C09138=1192.956,372.415,-78.592,-176.020,8.369,148.494
C09139=1192.960,372.168,-78.558,-176.022,8.366,148.494
C09140=1192.964,371.920,-78.523,-176.023,8.362,148.493
C09141=1192.968,371.672,-78.490,-176.024,8.359,148.493
C09142=1192.973,371.425,-78.456,-176.026,8.355,148.492
C09143=1192.976,371.177,-78.422,-176.027,8.353,148.492
C09144=1192.981,370.930,-78.387,-176.029,8.349,148.491
C09145=1192.985,370.683,-78.353,-176.030,8.346,148.491
C09146=1192.989,370.434,-78.318,-176.032,8.342,148.490
C09147=1192.993,370.187,-78.285,-176.033,8.339,148.490
C09148=1192.997,369.939,-78.251,-176.035,8.336,148.490
C09149=1193.000,369.692,-78.217,-176.036,8.333,148.489
C09150=1193.005,369.444,-78.182,-176.038,8.329,148.489
C09151=1193.009,369.196,-78.149,-176.039,8.327,148.488
C09152=1193.013,368.948,-78.114,-176.041,8.323,148.488
C09153=1193.017,368.701,-78.080,-176.042,8.320,148.488
C09154=1193.021,368.454,-78.046,-176.044,8.317,148.487
C09155=1193.025,368.205,-78.012,-176.045,8.314,148.487
C09156=1193.029,367.958,-77.978,-176.047,8.310,148.486
C09157=1193.033,367.711,-77.944,-176.048,8.307,148.486
C09158=1193.037,367.462,-77.910,-176.050,8.304,148.485
C09159=1193.042,367.215,-77.876,-176.051,8.300,148.485
C09160=1193.045,366.968,-77.842,-176.053,8.297,148.485
C09161=1193.050,366.686,-77.804,-176.054,8.294,148.484
C09162=1193.055,366.405,-77.765,-176.056,8.290,148.484
C09163=1193.059,366.125,-77.727,-176.059,8.285,148.483
C09164=1193.063,365.843,-77.688,-176.060,8.282,148.483
C09165=1193.068,365.596,-77.655,-176.062,8.279,148.482
C09166=1193.072,365.348,-77.620,-176.063,8.275,148.482
C09167=1193.075,365.100,-77.586,-176.065,8.272,148.482
C09168=1193.080,364.853,-77.553,-176.066,8.269,148.481
C09169=1193.084,364.605,-77.519,-176.069,8.266,148.481
C09170=1193.088,364.357,-77.485,-176.070,8.262,148.481
C09171=1193.092,364.110,-77.451,-176.072,8.259,148.480
C09172=1193.096,363.862,-77.417,-176.074,8.256,148.480
C09173=1193.100,363.615,-77.384,-176.075,8.252,148.479
C09174=1193.104,363.367,-77.350,-176.077,8.249,148.479
C09175=1193.108,363.119,-77.316,-176.079,8.246,148.479
C09176=1193.112,362.871,-77.282,-176.081,8.242,148.478
C09177=1193.116,362.624,-77.249,-176.082,8.240,148.478
C09178=1193.120,362.376,-77.215,-176.084,8.236,148.478
C09179=1193.124,362.129,-77.182,-176.086,8.232,148.477
C09180=1193.129,361.880,-77.147,-176.088,8.229,148.477
C09181=1193.133,361.633,-77.114,-176.089,8.226,148.477
C09182=1193.136,361.385,-77.080,-176.091,8.223,148.476
C09183=1193.141,361.138,-77.047,-176.093,8.219,148.476
C09184=1193.145,360.890,-77.013,-176.095,8.217,148.476
C09185=1193.149,360.642,-76.979,-176.096,8.213,148.475
C09186=1193.153,360.394,-76.946,-176.099,8.210,148.475
C09187=1193.157,360.147,-76.912,-176.100,8.206,148.474
C09188=1193.161,359.899,-76.879,-176.103,8.203,148.474
C09189=1193.166,359.651,-76.845,-176.104,8.200,148.474
C09190=1193.169,359.403,-76.811,-176.106,8.196,148.473
C09191=1193.173,359.156,-76.778,-176.108,8.193,148.473
C09192=1193.177,358.908,-76.745,-176.110,8.189,148.473
C09193=1193.181,358.660,-76.712,-176.111,8.187,148.473
C09194=1193.185,358.413,-76.678,-176.113,8.183,148.472
C09195=1193.189,358.165,-76.645,-176.115,8.180,148.472
C09196=1193.194,357.917,-76.611,-176.118,8.176,148.472
C09197=1193.198,357.669,-76.577,-176.119,8.173,148.471
C09198=1193.202,357.422,-76.543,-176.121,8.170,148.471
C09199=1193.206,357.174,-76.510,-176.123,8.167,148.471
C09200=1193.210,356.926,-76.477,-176.125,8.163,148.470
C09201=1193.214,356.679,-76.444,-176.127,8.160,148.470
C09202=1193.218,356.431,-76.411,-176.129,8.156,148.470
C09203=1193.222,356.183,-76.378,-176.131,8.154,148.470
C09204=1193.226,355.936,-76.344,-176.133,8.150,148.469
C09205=1193.230,355.688,-76.310,-176.135,8.147,148.469
C09206=1193.234,355.440,-76.277,-176.137,8.143,148.468
C09207=1193.239,355.192,-76.243,-176.139,8.140,148.468
C09208=1193.243,354.944,-76.210,-176.141,8.137,148.468
C09209=1193.247,354.696,-76.177,-176.142,8.134,148.468
C09210=1193.251,354.449,-76.144,-176.145,8.131,148.467
C09211=1193.255,354.201,-76.111,-176.147,8.127,148.467
C09212=1193.259,353.953,-76.078,-176.149,8.124,148.467
C09213=1193.263,353.705,-76.044,-176.151,8.120,148.466
C09214=1193.268,353.458,-76.011,-176.153,8.118,148.466
C09215=1193.272,353.210,-75.978,-176.155,8.114,148.466
C09216=1193.276,352.962,-75.945,-176.157,8.111,148.466
C09217=1193.280,352.715,-75.912,-176.159,8.107,148.465
C09218=1193.284,352.467,-75.879,-176.161,8.104,148.465
C09219=1193.288,352.219,-75.846,-176.163,8.102,148.465
C09220=1193.292,351.972,-75.813,-176.165,8.098,148.465
C09221=1193.296,351.724,-75.780,-176.167,8.095,148.464
C09222=1193.300,351.476,-75.747,-176.169,8.091,148.464
C09223=1193.304,351.228,-75.713,-176.171,8.088,148.464
C09224=1193.308,350.981,-75.680,-176.173,8.086,148.464
C09225=1193.312,350.733,-75.647,-176.175,8.082,148.464
C09226=1193.317,350.485,-75.614,-176.177,8.079,148.463
C09227=1193.321,350.237,-75.582,-176.179,8.075,148.463
C09228=1193.325,349.989,-75.548,-176.181,8.072,148.463
C09229=1193.329,349.741,-75.515,-176.184,8.069,148.462
C09230=1193.333,349.494,-75.482,-176.185,8.066,148.462
C09231=1193.337,349.246,-75.450,-176.188,8.063,148.462
C09232=1193.341,348.999,-75.416,-176.190,8.059,148.462
C09233=1193.345,348.750,-75.384,-176.192,8.056,148.461
C09234=1193.350,348.503,-75.351,-176.194,8.052,148.461
C09235=1193.354,348.255,-75.318,-176.195,8.050,148.461
C09236=1193.358,348.007,-75.284,-176.198,8.047,148.461
C09237=1193.362,347.759,-75.252,-176.200,8.043,148.461
C09238=1193.366,347.511,-75.219,-176.202,8.040,148.460
C09239=1193.370,347.264,-75.186,-176.204,8.037,148.460
C09240=1193.374,347.016,-75.153,-176.207,8.033,148.460
C09241=1193.378,346.768,-75.121,-176.208,8.031,148.460
C09242=1193.383,346.520,-75.088,-176.211,8.027,148.459
C09243=1193.386,346.272,-75.055,-176.213,8.024,148.459
C09244=1193.390,346.024,-75.023,-176.215,8.021,148.459
C09245=1193.395,345.777,-74.990,-176.217,8.017,148.459
C09246=1193.400,345.529,-74.957,-176.219,8.015,148.459
C09247=1193.403,345.281,-74.925,-176.221,8.012,148.458
C09248=1193.407,345.033,-74.892,-176.223,8.008,148.458
C09249=1193.412,344.785,-74.859,-176.226,8.005,148.458
C09250=1193.416,344.537,-74.826,-176.228,8.002,148.458
C09251=1193.419,344.289,-74.794,-176.230,7.998,148.458
C09252=1193.423,344.042,-74.761,-176.232,7.996,148.457
C09253=1193.428,343.793,-74.729,-176.234,7.993,148.457
C09254=1193.432,343.547,-74.696,-176.236,7.989,148.457
C09255=1193.436,343.298,-74.664,-176.239,7.986,148.457
C09256=1193.441,343.050,-74.631,-176.241,7.983,148.456
C09257=1193.445,342.802,-74.598,-176.242,7.980,148.456
C09258=1193.448,342.555,-74.566,-176.245,7.977,148.456
C09259=1193.453,342.306,-74.533,-176.247,7.973,148.456
C09260=1193.458,342.059,-74.501,-176.250,7.970,148.456
C09261=1193.461,341.811,-74.469,-176.252,7.967,148.456
C09262=1193.465,341.564,-74.436,-176.254,7.965,148.455
C09263=1193.469,341.316,-74.404,-176.256,7.961,148.455
C09264=1193.473,341.068,-74.371,-176.258,7.958,148.455
C09265=1193.478,340.789,-74.335,-176.260,7.955,148.455
C09266=1193.483,340.511,-74.299,-176.263,7.950,148.455
C09267=1193.488,340.232,-74.262,-176.266,7.947,148.455
C09268=1193.492,339.954,-74.225,-176.268,7.944,148.454
C09269=1193.496,339.705,-74.193,-176.270,7.941,148.454
C09270=1193.500,339.457,-74.161,-176.272,7.937,148.454
C09271=1193.504,339.210,-74.128,-176.275,7.934,148.454
C09272=1193.509,338.962,-74.096,-176.277,7.931,148.454
C09273=1193.513,338.714,-74.064,-176.279,7.929,148.453
C09274=1193.517,338.466,-74.031,-176.281,7.925,148.453
C09275=1193.521,338.218,-73.999,-176.284,7.922,148.453
C09276=1193.526,337.970,-73.967,-176.286,7.919,148.453
C09277=1193.530,337.722,-73.935,-176.288,7.916,148.453
C09278=1193.534,337.475,-73.902,-176.290,7.913,148.453
C09279=1193.537,337.227,-73.870,-176.292,7.910,148.452
C09280=1193.543,336.979,-73.838,-176.295,7.906,148.452
C09281=1193.546,336.731,-73.806,-176.297,7.903,148.452
C09282=1193.551,336.483,-73.774,-176.300,7.900,148.452
C09283=1193.554,336.235,-73.742,-176.301,7.898,148.452
C09284=1193.558,335.988,-73.710,-176.303,7.894,148.452
C09285=1193.563,335.739,-73.677,-176.306,7.891,148.452
C09286=1193.567,335.491,-73.645,-176.308,7.888,148.451
C09287=1193.571,335.243,-73.613,-176.311,7.885,148.451
C09288=1193.575,334.996,-73.581,-176.313,7.882,148.451
C09289=1193.580,334.747,-73.549,-176.315,7.879,148.451
C09290=1193.583,334.499,-73.517,-176.317,7.876,148.451
C09291=1193.588,334.252,-73.486,-176.320,7.872,148.451
C09292=1193.592,334.004,-73.453,-176.322,7.869,148.451
C09293=1193.596,333.756,-73.421,-176.324,7.866,148.450
C09294=1193.600,333.508,-73.390,-176.326,7.864,148.450
C09295=1193.605,333.260,-73.358,-176.329,7.860,148.450
C09296=1193.608,333.012,-73.326,-176.331,7.857,148.450
C09297=1193.613,332.764,-73.294,-176.334,7.854,148.450
C09298=1193.617,332.516,-73.262,-176.336,7.851,148.450
C09299=1193.621,332.268,-73.230,-176.338,7.848,148.450
C09300=1193.626,332.021,-73.198,-176.340,7.845,148.450
C09301=1193.630,331.773,-73.166,-176.343,7.842,148.449
C09302=1193.633,331.524,-73.134,-176.345,7.839,148.449
C09303=1193.638,331.277,-73.103,-176.348,7.836,148.449
C09304=1193.642,331.029,-73.070,-176.349,7.833,148.449
C09305=1193.646,330.781,-73.038,-176.352,7.830,148.449
C09306=1193.650,330.533,-73.007,-176.354,7.827,148.449
C09307=1193.654,330.285,-72.974,-176.356,7.823,148.449
C09308=1193.659,330.037,-72.944,-176.359,7.820,148.449
C09309=1193.663,329.789,-72.912,-176.361,7.817,148.448
C09310=1193.666,329.541,-72.880,-176.363,7.815,148.448
C09311=1193.672,329.293,-72.848,-176.366,7.812,148.448
C09312=1193.675,329.045,-72.816,-176.368,7.809,148.448
C09313=1193.680,328.797,-72.785,-176.371,7.805,148.448
C09314=1193.684,328.549,-72.753,-176.373,7.802,148.448
C09315=1193.687,328.301,-72.722,-176.375,7.800,148.448
C09316=1193.692,328.054,-72.690,-176.377,7.796,148.448
C09317=1193.696,327.805,-72.658,-176.380,7.793,148.448
C09318=1193.701,327.558,-72.627,-176.382,7.790,148.447
C09319=1193.704,327.310,-72.595,-176.385,7.787,148.447
C09320=1193.709,327.062,-72.564,-176.387,7.785,148.447
C09321=1193.713,326.814,-72.532,-176.389,7.782,148.447
C09322=1193.718,326.566,-72.500,-176.391,7.778,148.447
C09323=1193.721,326.318,-72.469,-176.394,7.775,148.447
C09324=1193.725,326.069,-72.437,-176.396,7.772,148.447
C09325=1193.730,325.822,-72.406,-176.399,7.770,148.447
C09326=1193.734,325.573,-72.375,-176.401,7.766,148.447
C09327=1193.738,325.326,-72.343,-176.403,7.763,148.447
C09328=1193.742,325.078,-72.311,-176.406,7.760,148.446
C09329=1193.746,324.830,-72.281,-176.408,7.757,148.446
C09330=1193.750,324.582,-72.249,-176.410,7.754,148.446
C09331=1193.755,324.334,-72.218,-176.413,7.751,148.446
C09332=1193.759,324.086,-72.186,-176.415,7.748,148.446
C09333=1193.764,323.838,-72.155,-176.418,7.745,148.446
C09334=1193.767,323.590,-72.123,-176.420,7.743,148.446
C09335=1193.772,323.342,-72.092,-176.422,7.740,148.446
C09336=1193.776,323.094,-72.060,-176.425,7.737,148.446
C09337=1193.780,322.846,-72.029,-176.427,7.733,148.446
C09338=1193.784,322.598,-71.998,-176.430,7.730,148.446
C09339=1193.789,322.350,-71.967,-176.432,7.728,148.446
C09340=1193.792,322.102,-71.935,-176.434,7.725,148.446
C09341=1193.797,321.854,-71.904,-176.437,7.722,148.446
C09342=1193.801,321.606,-71.873,-176.439,7.718,148.445
C09343=1193.805,321.358,-71.842,-176.442,7.715,148.445
C09344=1193.810,321.110,-71.810,-176.444,7.713,148.445
C09345=1193.814,320.862,-71.779,-176.446,7.710,148.445
C09346=1193.818,320.614,-71.749,-176.449,7.707,148.445
C09347=1193.821,320.366,-71.717,-176.451,7.704,148.445
C09348=1193.826,320.118,-71.686,-176.453,7.701,148.445
C09349=1193.830,319.869,-71.655,-176.456,7.698,148.445
C09350=1193.834,319.622,-71.624,-176.458,7.695,148.445
C09351=1193.839,319.374,-71.593,-176.461,7.692,148.445
C09352=1193.843,319.125,-71.562,-176.464,7.689,148.445
C09353=1193.847,318.878,-71.531,-176.465,7.686,148.445
C09354=1193.851,318.629,-71.499,-176.468,7.683,148.445
C09355=1193.856,318.381,-71.469,-176.470,7.680,148.444
C09356=1193.860,318.133,-71.438,-176.473,7.677,148.444
C09357=1193.864,317.885,-71.407,-176.476,7.674,148.444
C09358=1193.868,317.638,-71.376,-176.477,7.672,148.444
C09359=1193.873,317.390,-71.345,-176.480,7.669,148.444
C09360=1193.877,317.141,-71.314,-176.483,7.666,148.444
C09361=1193.881,316.893,-71.283,-176.485,7.663,148.444
C09362=1193.885,316.645,-71.252,-176.487,7.660,148.444
C09363=1193.889,316.398,-71.221,-176.490,7.657,148.444
C09364=1193.893,316.150,-71.190,-176.492,7.654,148.444
C09365=1193.897,315.901,-71.159,-176.495,7.651,148.444
C09366=1193.902,315.653,-71.129,-176.497,7.649,148.444
C09367=1193.907,315.405,-71.098,-176.499,7.645,148.444
C09368=1193.910,315.157,-71.067,-176.502,7.642,148.444
C09369=1193.915,314.881,-71.032,-176.504,7.639,148.444
C09370=1193.920,314.603,-70.998,-176.507,7.636,148.444
C09371=1193.925,314.328,-70.964,-176.510,7.632,148.444
C09372=1193.929,314.052,-70.930,-176.513,7.629,148.444
C09373=1193.933,313.803,-70.899,-176.515,7.626,148.444
C09374=1193.937,313.556,-70.869,-176.517,7.624,148.444
C09375=1193.942,313.308,-70.838,-176.520,7.621,148.444
C09376=1193.946,313.059,-70.807,-176.523,7.618,148.444
C09377=1193.951,312.811,-70.776,-176.525,7.614,148.444
C09378=1193.954,312.563,-70.746,-176.527,7.612,148.444
C09379=1193.959,312.315,-70.715,-176.530,7.609,148.444
C09380=1193.963,312.067,-70.684,-176.533,7.606,148.444
C09381=1193.967,311.818,-70.654,-176.535,7.603,148.443
C09382=1193.972,311.570,-70.624,-176.537,7.601,148.443
C09383=1193.976,311.323,-70.593,-176.540,7.598,148.443
C09384=1193.980,311.074,-70.562,-176.542,7.595,148.443
C09385=1193.984,310.826,-70.532,-176.545,7.591,148.443
C09386=1193.988,310.579,-70.501,-176.547,7.589,148.443
C09387=1193.993,310.331,-70.471,-176.549,7.586,148.443
C09388=1193.997,310.082,-70.439,-176.552,7.583,148.443
C09389=1194.001,309.834,-70.410,-176.555,7.580,148.443
C09390=1194.006,309.586,-70.379,-176.557,7.578,148.443
C09391=1194.010,309.338,-70.349,-176.559,7.575,148.443
C09392=1194.014,309.090,-70.318,-176.562,7.572,148.443
C09393=1194.018,308.841,-70.288,-176.565,7.569,148.443
C09394=1194.022,308.593,-70.258,-176.567,7.566,148.443
C09395=1194.027,308.345,-70.227,-176.569,7.563,148.443
C09396=1194.031,308.098,-70.197,-176.572,7.560,148.443
C09397=1194.036,307.849,-70.167,-176.574,7.557,148.443
C09398=1194.039,307.601,-70.136,-176.577,7.555,148.443
C09399=1194.044,307.353,-70.105,-176.579,7.552,148.443
C09400=1194.048,307.104,-70.076,-176.582,7.549,148.443
C09401=1194.052,306.856,-70.045,-176.584,7.545,148.443
C09402=1194.056,306.609,-70.015,-176.586,7.543,148.443
C09403=1194.061,306.360,-69.985,-176.589,7.540,148.443
C09404=1194.065,306.113,-69.955,-176.592,7.537,148.443
C09405=1194.069,305.864,-69.924,-176.594,7.534,148.443
C09406=1194.073,305.616,-69.894,-176.597,7.532,148.443
C09407=1194.078,305.368,-69.864,-176.599,7.529,148.443
C09408=1194.082,305.119,-69.834,-176.602,7.526,148.443
C09409=1194.087,304.871,-69.803,-176.604,7.524,148.443
C09410=1194.091,304.623,-69.774,-176.606,7.521,148.443
C09411=1194.095,304.375,-69.743,-176.609,7.518,148.443
C09412=1194.099,304.128,-69.713,-176.612,7.515,148.443
C09413=1194.104,303.879,-69.683,-176.614,7.512,148.443
C09414=1194.108,303.631,-69.652,-176.617,7.509,148.443
C09415=1194.112,303.382,-69.623,-176.619,7.506,148.443
C09416=1194.116,303.134,-69.592,-176.622,7.503,148.443
C09417=1194.121,302.886,-69.563,-176.624,7.501,148.443
C09418=1194.125,302.638,-69.533,-176.626,7.498,148.443
C09419=1194.129,302.390,-69.502,-176.629,7.495,148.443
C09420=1194.134,302.142,-69.473,-176.631,7.493,148.443
C09421=1194.137,301.894,-69.443,-176.634,7.490,148.443
C09422=1194.142,301.645,-69.413,-176.637,7.487,148.443
C09423=1194.146,301.397,-69.383,-176.639,7.484,148.443
C09424=1194.150,301.150,-69.353,-176.642,7.481,148.443
C09425=1194.155,300.901,-69.323,-176.644,7.478,148.443
C09426=1194.159,300.653,-69.293,-176.647,7.475,148.443
C09427=1194.163,300.405,-69.263,-176.649,7.473,148.443
C09428=1194.168,300.156,-69.233,-176.651,7.470,148.443
C09429=1194.172,299.908,-69.204,-176.654,7.467,148.443
C09430=1194.176,299.661,-69.174,-176.656,7.465,148.443
C09431=1194.180,299.412,-69.144,-176.659,7.462,148.443
C09432=1194.185,299.164,-69.114,-176.662,7.459,148.443
C09433=1194.189,298.916,-69.084,-176.664,7.456,148.443
C09434=1194.193,298.668,-69.055,-176.666,7.453,148.443
C09435=1194.198,298.420,-69.025,-176.669,7.450,148.443
C09436=1194.203,298.171,-68.995,-176.672,7.447,148.443
C09437=1194.206,297.923,-68.965,-176.674,7.445,148.444
C09438=1194.211,297.675,-68.936,-176.677,7.442,148.444
C09439=1194.215,297.427,-68.906,-176.679,7.439,148.444
C09440=1194.219,297.179,-68.877,-176.682,7.437,148.444
C09441=1194.224,296.930,-68.847,-176.684,7.434,148.444
C09442=1194.228,296.682,-68.817,-176.687,7.431,148.444
C09443=1194.232,296.434,-68.787,-176.690,7.428,148.444
C09444=1194.236,296.186,-68.758,-176.692,7.426,148.444
C09445=1194.240,295.938,-68.728,-176.694,7.423,148.444
C09446=1194.245,295.689,-68.699,-176.697,7.420,148.444
C09447=1194.249,295.441,-68.669,-176.699,7.418,148.444
C09448=1194.254,295.192,-68.639,-176.702,7.415,148.444
C09449=1194.258,294.944,-68.610,-176.705,7.412,148.444
C09450=1194.262,294.696,-68.580,-176.707,7.409,148.444
C09451=1194.266,294.448,-68.551,-176.710,7.406,148.444
C09452=1194.270,294.199,-68.521,-176.712,7.403,148.444
C09453=1194.275,293.952,-68.492,-176.714,7.401,148.444
C09454=1194.279,293.703,-68.463,-176.717,7.398,148.444
C09455=1194.283,293.455,-68.433,-176.720,7.395,148.444
C09456=1194.288,293.207,-68.404,-176.722,7.393,148.444
C09457=1194.292,292.959,-68.374,-176.725,7.390,148.444
C09458=1194.296,292.710,-68.345,-176.727,7.387,148.444
C09459=1194.300,292.462,-68.316,-176.730,7.385,148.444
C09460=1194.304,292.214,-68.286,-176.732,7.382,148.444
C09461=1194.309,291.966,-68.257,-176.735,7.379,148.444
C09462=1194.313,291.718,-68.228,-176.737,7.377,148.444
C09463=1194.318,291.470,-68.198,-176.740,7.374,148.444
C09464=1194.322,291.221,-68.169,-176.743,7.371,148.444
C09465=1194.326,290.973,-68.140,-176.745,7.369,148.445
C09466=1194.330,290.724,-68.110,-176.747,7.365,148.445
C09467=1194.335,290.476,-68.081,-176.750,7.362,148.445
C09468=1194.339,290.229,-68.052,-176.752,7.360,148.445
C09469=1194.344,289.980,-68.022,-176.755,7.357,148.445
C09470=1194.348,289.731,-67.994,-176.758,7.354,148.445
C09471=1194.352,289.483,-67.964,-176.760,7.352,148.445
C09472=1194.356,289.235,-67.935,-176.763,7.349,148.445
C09473=1194.361,288.960,-67.903,-176.765,7.346,148.445
C09474=1194.366,288.686,-67.870,-176.768,7.343,148.445
C09475=1194.371,288.411,-67.838,-176.771,7.340,148.445
C09476=1194.375,288.137,-67.807,-176.774,7.337,148.445
C09477=1194.380,287.889,-67.777,-176.777,7.334,148.445
C09478=1194.384,287.640,-67.748,-176.779,7.332,148.445
C09479=1194.389,287.392,-67.719,-176.781,7.329,148.445
C09480=1194.393,287.144,-67.690,-176.784,7.326,148.445
C09481=1194.397,286.896,-67.660,-176.786,7.324,148.445
C09482=1194.401,286.647,-67.632,-176.789,7.321,148.445
C09483=1194.406,286.400,-67.603,-176.792,7.318,148.446
C09484=1194.410,286.151,-67.574,-176.794,7.316,148.446
C09485=1194.414,285.902,-67.545,-176.797,7.313,148.446
C09486=1194.419,285.654,-67.515,-176.799,7.311,148.446
C09487=1194.424,285.406,-67.487,-176.802,7.308,148.446
C09488=1194.427,285.158,-67.458,-176.805,7.305,148.446
C09489=1194.432,284.909,-67.430,-176.807,7.303,148.446
C09490=1194.436,284.662,-67.400,-176.809,7.300,148.446
C09491=1194.441,284.413,-67.371,-176.812,7.297,148.446
C09492=1194.444,284.165,-67.343,-176.814,7.295,148.446
C09493=1194.449,283.916,-67.313,-176.817,7.292,148.446
C09494=1194.454,283.668,-67.285,-176.820,7.290,148.446
C09495=1194.458,283.419,-67.256,-176.822,7.287,148.446
C09496=1194.462,283.171,-67.227,-176.825,7.284,148.446
C09497=1194.467,282.923,-67.199,-176.827,7.282,148.447
C09498=1194.471,282.675,-67.170,-176.830,7.279,148.447
C09499=1194.475,282.426,-67.141,-176.832,7.276,148.447
C09500=1194.479,282.179,-67.112,-176.835,7.273,148.447
C09501=1194.484,281.930,-67.084,-176.838,7.271,148.447
C09502=1194.488,281.681,-67.055,-176.840,7.268,148.447
C09503=1194.492,281.434,-67.026,-176.843,7.265,148.447
C09504=1194.497,281.185,-66.998,-176.845,7.262,148.447
C09505=1194.501,280.937,-66.968,-176.848,7.260,148.447
C09506=1194.505,280.689,-66.940,-176.850,7.257,148.447
C09507=1194.510,280.440,-66.912,-176.852,7.255,148.447
C09508=1194.514,280.192,-66.882,-176.856,7.252,148.447
C09509=1194.518,279.944,-66.854,-176.858,7.249,148.448
C09510=1194.523,279.695,-66.826,-176.860,7.247,148.448
C09511=1194.527,279.447,-66.798,-176.863,7.244,148.448
C09512=1194.531,279.199,-66.768,-176.865,7.242,148.448
C09513=1194.536,278.950,-66.740,-176.868,7.239,148.448
C09514=1194.540,278.702,-66.712,-176.871,7.237,148.448
C09515=1194.545,278.453,-66.683,-176.873,7.234,148.448
C09516=1194.548,278.205,-66.654,-176.876,7.231,148.448
C09517=1194.553,277.957,-66.626,-176.878,7.229,148.448
C09518=1194.557,277.708,-66.598,-176.881,7.226,148.448
C09519=1194.562,277.460,-66.569,-176.884,7.224,148.449
C09520=1194.566,277.212,-66.541,-176.886,7.221,148.449
C09521=1194.571,276.963,-66.513,-176.889,7.218,148.449
C09522=1194.574,276.715,-66.484,-176.891,7.216,148.449
C09523=1194.579,276.467,-66.455,-176.894,7.213,148.449
C09524=1194.583,276.219,-66.428,-176.896,7.211,148.449
C09525=1194.588,275.970,-66.399,-176.899,7.208,148.449
C09526=1194.592,275.722,-66.371,-176.901,7.206,148.449
C09527=1194.597,275.473,-66.342,-176.904,7.203,148.449
C09528=1194.601,275.225,-66.315,-176.906,7.201,148.449
C09529=1194.605,274.976,-66.286,-176.909,7.198,148.449
C09530=1194.610,274.728,-66.258,-176.912,7.195,148.450
C09531=1194.614,274.479,-66.229,-176.914,7.193,148.450
C09532=1194.619,274.232,-66.202,-176.917,7.190,148.450
C09533=1194.623,273.983,-66.173,-176.919,7.188,148.450
C09534=1194.627,273.735,-66.145,-176.922,7.185,148.450
C09535=1194.631,273.486,-66.117,-176.924,7.183,148.450
C09536=1194.636,273.238,-66.088,-176.927,7.180,148.450
C09537=1194.640,272.990,-66.060,-176.929,7.178,148.450
C09538=1194.645,272.741,-66.032,-176.932,7.175,148.450
C09539=1194.649,272.493,-66.004,-176.935,7.172,148.450
C09540=1194.653,272.245,-65.976,-176.937,7.170,148.451
C09541=1194.658,271.996,-65.947,-176.940,7.167,148.451
C09542=1194.662,271.748,-65.920,-176.942,7.165,148.451
C09543=1194.666,271.500,-65.891,-176.945,7.162,148.451
C09544=1194.671,271.251,-65.863,-176.948,7.160,148.451
C09545=1194.675,271.002,-65.836,-176.950,7.157,148.451
C09546=1194.679,270.754,-65.808,-176.952,7.155,148.451
C09547=1194.684,270.505,-65.779,-176.956,7.152,148.451
C09548=1194.688,270.258,-65.751,-176.958,7.150,148.451
C09549=1194.693,270.010,-65.724,-176.960,7.147,148.452
C09550=1194.697,269.761,-65.695,-176.963,7.145,148.452
C09551=1194.702,269.512,-65.668,-176.966,7.142,148.452
C09552=1194.705,269.264,-65.640,-176.968,7.139,148.452
C09553=1194.710,269.015,-65.611,-176.971,7.137,148.452
C09554=1194.715,268.768,-65.583,-176.973,7.134,148.452
C09555=1194.719,268.518,-65.556,-176.976,7.132,148.452
C09556=1194.723,268.271,-65.528,-176.979,7.129,148.452
C09557=1194.728,268.022,-65.500,-176.981,7.127,148.452
C09558=1194.732,267.773,-65.472,-176.984,7.124,148.453
C09559=1194.737,267.525,-65.445,-176.986,7.122,148.453
C09560=1194.740,267.277,-65.417,-176.989,7.119,148.453
C09561=1194.745,267.028,-65.389,-176.991,7.117,148.453
C09562=1194.750,266.779,-65.361,-176.994,7.114,148.453
C09563=1194.754,266.531,-65.333,-176.996,7.112,148.453
C09564=1194.759,266.283,-65.306,-176.999,7.109,148.453
C09565=1194.762,266.034,-65.278,-177.002,7.107,148.454
C09566=1194.767,265.787,-65.250,-177.004,7.104,148.454
C09567=1194.772,265.538,-65.222,-177.007,7.102,148.454
C09568=1194.776,265.289,-65.194,-177.009,7.099,148.454
C09569=1194.781,265.041,-65.167,-177.012,7.097,148.454
C09570=1194.785,264.793,-65.139,-177.015,7.094,148.454
C09571=1194.789,264.544,-65.112,-177.017,7.092,148.454
C09572=1194.793,264.296,-65.084,-177.020,7.089,148.454
C09573=1194.798,264.047,-65.057,-177.022,7.087,148.455
C09574=1194.802,263.799,-65.029,-177.025,7.084,148.455
C09575=1194.807,263.550,-65.001,-177.027,7.082,148.455
C09576=1194.811,263.302,-64.973,-177.030,7.079,148.455
C09577=1194.815,263.029,-64.943,-177.032,7.077,148.455
C09578=1194.821,262.756,-64.913,-177.036,7.074,148.455
C09579=1194.826,262.484,-64.883,-177.038,7.071,148.455
C09580=1194.830,262.211,-64.853,-177.041,7.069,148.456
C09581=1194.834,261.962,-64.826,-177.044,7.066,148.456
C09582=1194.839,261.714,-64.799,-177.046,7.064,148.456
C09583=1194.844,261.465,-64.770,-177.049,7.062,148.456
C09584=1194.848,261.216,-64.743,-177.052,7.059,148.456
C09585=1194.853,260.968,-64.715,-177.054,7.056,148.456
C09586=1194.857,260.720,-64.688,-177.057,7.054,148.456
C09587=1194.861,260.471,-64.661,-177.059,7.052,148.457
C09588=1194.866,260.223,-64.633,-177.062,7.049,148.457
C09589=1194.870,259.974,-64.606,-177.064,7.047,148.457
C09590=1194.874,259.726,-64.579,-177.067,7.045,148.457
C09591=1194.879,259.478,-64.552,-177.070,7.042,148.457
C09592=1194.883,259.229,-64.524,-177.072,7.040,148.457
C09593=1194.887,258.981,-64.497,-177.075,7.037,148.457
C09594=1194.892,258.732,-64.470,-177.077,7.035,148.458
C09595=1194.896,258.484,-64.442,-177.080,7.032,148.458
C09596=1194.900,258.235,-64.415,-177.082,7.030,148.458
C09597=1194.905,257.987,-64.388,-177.085,7.027,148.458
C09598=1194.910,257.738,-64.361,-177.088,7.025,148.458
C09599=1194.914,257.490,-64.333,-177.090,7.022,148.458
C09600=1194.919,257.242,-64.306,-177.093,7.020,148.459
C09601=1194.923,256.993,-64.279,-177.095,7.018,148.459
C09602=1194.927,256.744,-64.251,-177.098,7.015,148.459
C09603=1194.931,256.496,-64.225,-177.100,7.013,148.459
C09604=1194.936,256.247,-64.198,-177.103,7.010,148.459
C09605=1194.941,255.999,-64.171,-177.106,7.008,148.459
C09606=1194.945,255.750,-64.144,-177.108,7.005,148.459
C09607=1194.950,255.502,-64.117,-177.111,7.003,148.460
C09608=1194.954,255.253,-64.088,-177.113,7.001,148.460
C09609=1194.958,255.005,-64.062,-177.116,6.998,148.460
C09610=1194.962,254.757,-64.035,-177.119,6.996,148.460
C09611=1194.967,254.508,-64.008,-177.121,6.993,148.460
C09612=1194.972,254.260,-63.981,-177.124,6.992,148.461
C09613=1194.976,254.011,-63.954,-177.126,6.989,148.461
C09614=1194.980,253.763,-63.927,-177.129,6.986,148.461
C09615=1194.985,253.514,-63.900,-177.131,6.985,148.461
C09616=1194.989,253.265,-63.873,-177.134,6.982,148.461
C09617=1194.994,253.017,-63.846,-177.137,6.980,148.461
C09618=1194.997,252.768,-63.819,-177.140,6.977,148.461
C09619=1195.002,252.520,-63.792,-177.142,6.975,148.461
C09620=1195.007,252.272,-63.765,-177.144,6.973,148.462
C09621=1195.011,252.023,-63.738,-177.147,6.970,148.462
C09622=1195.016,251.774,-63.712,-177.150,6.968,148.462
C09623=1195.020,251.526,-63.685,-177.152,6.965,148.462
C09624=1195.025,251.277,-63.658,-177.155,6.963,148.463
C09625=1195.030,251.029,-63.631,-177.157,6.961,148.463
C09626=1195.034,250.781,-63.605,-177.160,6.958,148.463
C09627=1195.038,250.532,-63.578,-177.162,6.956,148.463
C09628=1195.043,250.284,-63.550,-177.165,6.953,148.463
C09629=1195.046,250.035,-63.524,-177.168,6.951,148.463
C09630=1195.051,249.786,-63.497,-177.170,6.949,148.463
C09631=1195.056,249.537,-63.470,-177.173,6.946,148.464
C09632=1195.060,249.289,-63.444,-177.175,6.944,148.464
C09633=1195.064,249.040,-63.417,-177.178,6.942,148.464
C09634=1195.068,248.792,-63.390,-177.181,6.939,148.464
C09635=1195.073,248.543,-63.364,-177.183,6.938,148.464
C09636=1195.078,248.295,-63.337,-177.186,6.935,148.465
C09637=1195.082,248.046,-63.310,-177.188,6.932,148.465
C09638=1195.087,247.798,-63.283,-177.191,6.931,148.465
C09639=1195.091,247.549,-63.258,-177.194,6.928,148.465
C09640=1195.095,247.301,-63.230,-177.196,6.926,148.465
C09641=1195.100,247.052,-63.203,-177.198,6.924,148.465
C09642=1195.104,246.803,-63.178,-177.202,6.921,148.466
C09643=1195.109,246.555,-63.151,-177.204,6.919,148.466
C09644=1195.113,246.307,-63.124,-177.206,6.917,148.466
C09645=1195.118,246.057,-63.098,-177.209,6.914,148.466
C09646=1195.122,245.809,-63.071,-177.212,6.912,148.466
C09647=1195.126,245.561,-63.044,-177.214,6.909,148.467
C09648=1195.131,245.313,-63.019,-177.217,6.907,148.467
C09649=1195.136,245.064,-62.992,-177.219,6.905,148.467
C09650=1195.140,244.815,-62.966,-177.222,6.902,148.467
C09651=1195.145,244.567,-62.939,-177.225,6.900,148.467
C09652=1195.149,244.318,-62.913,-177.227,6.898,148.468
C09653=1195.154,244.070,-62.886,-177.230,6.895,148.468
C09654=1195.158,243.821,-62.860,-177.233,6.894,148.468
C09655=1195.163,243.572,-62.833,-177.235,6.891,148.468
C09656=1195.166,243.324,-62.807,-177.238,6.889,148.468
C09657=1195.171,243.075,-62.781,-177.240,6.887,148.468
C09658=1195.175,242.827,-62.754,-177.243,6.885,148.469
C09659=1195.180,242.578,-62.728,-177.245,6.882,148.469
C09660=1195.185,242.329,-62.702,-177.248,6.880,148.469
C09661=1195.189,242.081,-62.676,-177.250,6.878,148.469
C09662=1195.194,241.832,-62.650,-177.253,6.875,148.470
C09663=1195.198,241.584,-62.623,-177.256,6.873,148.470
C09664=1195.203,241.335,-62.597,-177.258,6.871,148.470
C09665=1195.207,241.087,-62.570,-177.261,6.868,148.470
C09666=1195.211,240.838,-62.545,-177.264,6.866,148.470
C09667=1195.216,240.589,-62.518,-177.266,6.864,148.470
C09668=1195.220,240.341,-62.492,-177.269,6.861,148.471
C09669=1195.225,240.093,-62.466,-177.272,6.860,148.471
C09670=1195.230,239.843,-62.440,-177.274,6.857,148.471
C09671=1195.234,239.595,-62.414,-177.277,6.855,148.471
C09672=1195.238,239.347,-62.388,-177.279,6.853,148.472
C09673=1195.243,239.097,-62.361,-177.282,6.851,148.472
C09674=1195.247,238.849,-62.335,-177.284,6.848,148.472
C09675=1195.252,238.601,-62.310,-177.287,6.846,148.472
C09676=1195.256,238.352,-62.283,-177.289,6.844,148.472
C09677=1195.260,238.104,-62.257,-177.292,6.842,148.473
C09678=1195.265,237.855,-62.231,-177.295,6.839,148.473
C09679=1195.269,237.606,-62.205,-177.297,6.837,148.473
C09680=1195.274,237.358,-62.179,-177.300,6.835,148.473
C09681=1195.279,237.087,-62.151,-177.303,6.832,148.473
C09682=1195.284,236.815,-62.122,-177.306,6.830,148.474
C09683=1195.288,236.543,-62.094,-177.308,6.828,148.474
C09684=1195.294,236.272,-62.065,-177.312,6.825,148.474
C09685=1195.298,236.023,-62.040,-177.314,6.823,148.474
C09686=1195.302,235.774,-62.014,-177.316,6.821,148.475
C09687=1195.307,235.525,-61.988,-177.319,6.818,148.475
C09688=1195.311,235.278,-61.962,-177.322,6.816,148.475
C09689=1195.316,235.029,-61.936,-177.324,6.814,148.475
C09690=1195.320,234.780,-61.910,-177.327,6.812,148.476
C09691=1195.325,234.531,-61.884,-177.330,6.810,148.476
C09692=1195.329,234.283,-61.859,-177.332,6.808,148.476
C09693=1195.334,234.034,-61.833,-177.335,6.806,148.476
C09694=1195.338,233.785,-61.807,-177.337,6.803,148.476
C09695=1195.343,233.536,-61.781,-177.340,6.801,148.477
C09696=1195.348,233.288,-61.756,-177.343,6.799,148.477
C09697=1195.352,233.039,-61.730,-177.345,6.797,148.477
C09698=1195.356,232.791,-61.704,-177.348,6.794,148.477
C09699=1195.361,232.543,-61.679,-177.350,6.792,148.477
C09700=1195.365,232.294,-61.653,-177.353,6.790,148.478
C09701=1195.369,232.045,-61.627,-177.355,6.788,148.478
C09702=1195.374,231.797,-61.602,-177.358,6.785,148.478
C09703=1195.378,231.548,-61.576,-177.361,6.784,148.479
C09704=1195.383,231.299,-61.550,-177.363,6.782,148.479
C09705=1195.388,231.050,-61.524,-177.366,6.779,148.479
C09706=1195.392,230.802,-61.499,-177.369,6.777,148.479
C09707=1195.397,230.553,-61.473,-177.371,6.775,148.479
C09708=1195.401,230.304,-61.447,-177.374,6.773,148.480
C09709=1195.406,230.056,-61.422,-177.377,6.770,148.480
C09710=1195.410,229.807,-61.397,-177.379,6.768,148.480
C09711=1195.415,229.559,-61.371,-177.382,6.766,148.480
C09712=1195.419,229.310,-61.346,-177.384,6.765,148.481
C09713=1195.423,229.061,-61.320,-177.387,6.762,148.481
C09714=1195.428,228.813,-61.294,-177.390,6.760,148.481
C09715=1195.433,228.564,-61.269,-177.392,6.758,148.481
C09716=1195.437,228.315,-61.244,-177.394,6.756,148.482
C09717=1195.442,228.067,-61.218,-177.398,6.753,148.482
C09718=1195.446,227.818,-61.193,-177.400,6.751,148.482
C09719=1195.450,227.569,-61.167,-177.402,6.749,148.482
C09720=1195.455,227.321,-61.141,-177.405,6.747,148.483
C09721=1195.460,227.072,-61.116,-177.407,6.745,148.483
C09722=1195.465,226.823,-61.091,-177.411,6.742,148.483
C09723=1195.469,226.575,-61.065,-177.413,6.741,148.483
C09724=1195.472,226.326,-61.040,-177.415,6.738,148.483
C09725=1195.477,226.077,-61.015,-177.418,6.737,148.484
C09726=1195.482,225.829,-60.990,-177.421,6.734,148.484
C09727=1195.486,225.581,-60.964,-177.423,6.732,148.484
C09728=1195.491,225.331,-60.939,-177.426,6.730,148.485
C09729=1195.496,225.083,-60.914,-177.429,6.728,148.485
C09730=1195.500,224.834,-60.888,-177.432,6.726,148.485
C09731=1195.505,224.585,-60.863,-177.434,6.723,148.485
C09732=1195.509,224.337,-60.838,-177.437,6.722,148.486
C09733=1195.513,224.088,-60.813,-177.439,6.720,148.486
C09734=1195.518,223.839,-60.788,-177.441,6.718,148.486
C09735=1195.522,223.591,-60.762,-177.445,6.715,148.486
C09736=1195.527,223.342,-60.737,-177.447,6.713,148.487
C09737=1195.532,223.093,-60.712,-177.449,6.711,148.487
C09738=1195.537,222.844,-60.687,-177.452,6.709,148.487
C09739=1195.540,222.596,-60.662,-177.455,6.707,148.487
C09740=1195.545,222.347,-60.637,-177.457,6.704,148.487
C09741=1195.550,222.098,-60.611,-177.460,6.702,148.488
C09742=1195.555,221.850,-60.587,-177.463,6.701,148.488
C09743=1195.559,221.601,-60.561,-177.465,6.699,148.488
C09744=1195.563,221.352,-60.537,-177.468,6.697,148.489
C09745=1195.567,221.104,-60.511,-177.471,6.694,148.489
C09746=1195.573,220.855,-60.487,-177.473,6.692,148.489
C09747=1195.577,220.606,-60.461,-177.476,6.690,148.489
C09748=1195.581,220.358,-60.437,-177.478,6.688,148.490
C09749=1195.585,220.109,-60.411,-177.481,6.686,148.490
C09750=1195.591,219.860,-60.386,-177.484,6.684,148.490
C09751=1195.594,219.611,-60.362,-177.486,6.682,148.490
C09752=1195.599,219.363,-60.336,-177.489,6.680,148.491
C09753=1195.604,219.114,-60.311,-177.492,6.678,148.491
C09754=1195.609,218.865,-60.287,-177.494,6.676,148.491
C09755=1195.613,218.617,-60.262,-177.497,6.673,148.491
C09756=1195.617,218.368,-60.237,-177.500,6.671,148.492
C09757=1195.623,218.119,-60.212,-177.502,6.669,148.492
C09758=1195.626,217.870,-60.187,-177.505,6.668,148.492
C09759=1195.631,217.622,-60.162,-177.507,6.665,148.493
C09760=1195.636,217.372,-60.137,-177.510,6.663,148.493
C09761=1195.640,217.124,-60.113,-177.513,6.661,148.493
C09762=1195.645,216.876,-60.088,-177.516,6.659,148.494
C09763=1195.649,216.627,-60.063,-177.518,6.657,148.494
C09764=1195.654,216.378,-60.039,-177.520,6.655,148.494
C09765=1195.658,216.129,-60.013,-177.523,6.653,148.494
C09766=1195.663,215.881,-59.989,-177.526,6.651,148.495
C09767=1195.668,215.632,-59.964,-177.528,6.649,148.495
C09768=1195.671,215.383,-59.940,-177.531,6.647,148.495
C09769=1195.676,215.135,-59.914,-177.534,6.645,148.495
C09770=1195.681,214.885,-59.889,-177.536,6.643,148.496
C09771=1195.685,214.637,-59.865,-177.539,6.640,148.496
C09772=1195.690,214.388,-59.841,-177.542,6.638,148.496
C09773=1195.694,214.139,-59.816,-177.544,6.637,148.497
C09774=1195.699,213.890,-59.792,-177.547,6.635,148.497
C09775=1195.704,213.642,-59.768,-177.550,6.633,148.497
C09776=1195.708,213.393,-59.742,-177.552,6.631,148.497
C09777=1195.712,213.145,-59.718,-177.555,6.629,148.498
C09778=1195.717,212.896,-59.693,-177.558,6.626,148.498
C09779=1195.721,212.647,-59.669,-177.560,6.624,148.498
C09780=1195.726,212.398,-59.644,-177.563,6.622,148.498
C09781=1195.731,212.150,-59.620,-177.565,6.620,148.499
C09782=1195.735,211.900,-59.595,-177.568,6.619,148.499
C09783=1195.740,211.652,-59.571,-177.570,6.617,148.499
C09784=1195.745,211.403,-59.546,-177.574,6.614,148.500
C09785=1195.749,211.132,-59.519,-177.576,6.612,148.500
C09786=1195.754,210.862,-59.493,-177.579,6.611,148.500
C09787=1195.759,210.592,-59.467,-177.582,6.608,148.501
C09788=1195.764,210.321,-59.440,-177.584,6.606,148.501
C09789=1195.769,210.072,-59.415,-177.587,6.604,148.501
C09790=1195.773,209.824,-59.391,-177.590,6.602,148.501
C09791=1195.778,209.575,-59.367,-177.593,6.599,148.502
C09792=1195.783,209.326,-59.342,-177.596,6.598,148.502
C09793=1195.787,209.077,-59.318,-177.598,6.596,148.502
C09794=1195.792,208.829,-59.293,-177.600,6.594,148.503
C09795=1195.796,208.580,-59.269,-177.603,6.592,148.503
C09796=1195.801,208.332,-59.245,-177.606,6.590,148.503
C09797=1195.805,208.082,-59.221,-177.608,6.588,148.504
C09798=1195.810,207.833,-59.197,-177.612,6.586,148.504
C09799=1195.814,207.585,-59.173,-177.614,6.583,148.504
C09800=1195.819,207.336,-59.148,-177.616,6.582,148.504
C09801=1195.824,207.088,-59.124,-177.619,6.580,148.505
C09802=1195.827,206.839,-59.099,-177.622,6.578,148.505
C09803=1195.833,206.589,-59.075,-177.624,6.576,148.505
C09804=1195.837,206.341,-59.051,-177.627,6.574,148.506
C09805=1195.842,206.093,-59.027,-177.629,6.572,148.506
C09806=1195.847,205.844,-59.003,-177.632,6.570,148.506
C09807=1195.851,205.595,-58.978,-177.635,6.568,148.506
C09808=1195.855,205.346,-58.955,-177.638,6.566,148.507
C09809=1195.860,205.097,-58.930,-177.640,6.564,148.507
C09810=1195.865,204.849,-58.906,-177.643,6.562,148.508
C09811=1195.870,204.600,-58.883,-177.645,6.560,148.508
C09812=1195.873,204.350,-58.858,-177.648,6.558,148.508
C09813=1195.878,204.102,-58.834,-177.650,6.557,148.508
C09814=1195.883,203.853,-58.810,-177.653,6.555,148.509
C09815=1195.888,203.604,-58.786,-177.656,6.553,148.509
C09816=1195.892,203.356,-58.762,-177.658,6.551,148.509
C09817=1195.897,203.107,-58.739,-177.662,6.548,148.510
C09818=1195.901,202.857,-58.714,-177.664,6.546,148.510
C09819=1195.906,202.609,-58.690,-177.666,6.545,148.510
C09820=1195.910,202.360,-58.666,-177.669,6.543,148.510
C09821=1195.915,202.111,-58.642,-177.672,6.541,148.511
C09822=1195.919,201.862,-58.619,-177.674,6.539,148.511
C09823=1195.924,201.614,-58.595,-177.677,6.537,148.512
C09824=1195.929,201.365,-58.570,-177.680,6.535,148.512
C09825=1195.934,201.116,-58.547,-177.682,6.533,148.512
C09826=1195.937,200.867,-58.522,-177.685,6.531,148.512
C09827=1195.942,200.618,-58.499,-177.687,6.530,148.513
C09828=1195.946,200.370,-58.475,-177.690,6.528,148.513
C09829=1195.951,200.121,-58.452,-177.693,6.526,148.513
C09830=1195.956,199.872,-58.427,-177.696,6.523,148.514
C09831=1195.960,199.623,-58.404,-177.698,6.522,148.514
C09832=1195.965,199.375,-58.379,-177.701,6.520,148.514
C09833=1195.970,199.126,-58.356,-177.703,6.518,148.514
C09834=1195.975,198.877,-58.332,-177.706,6.516,148.515
C09835=1195.979,198.628,-58.309,-177.709,6.514,148.515
C09836=1195.984,198.380,-58.285,-177.711,6.512,148.516
C09837=1195.988,198.131,-58.261,-177.714,6.510,148.516
C09838=1195.993,197.882,-58.238,-177.717,6.509,148.516
C09839=1195.997,197.632,-58.213,-177.719,6.507,148.517
C09840=1196.001,197.383,-58.190,-177.722,6.505,148.517
C09841=1196.006,197.134,-58.167,-177.725,6.503,148.517
C09842=1196.011,196.886,-58.143,-177.727,6.501,148.517
C09843=1196.015,196.637,-58.119,-177.729,6.499,148.518
C09844=1196.020,196.389,-58.095,-177.732,6.497,148.518
C09845=1196.024,196.140,-58.072,-177.735,6.496,148.518
C09846=1196.029,195.890,-58.048,-177.737,6.494,148.519
C09847=1196.034,195.641,-58.025,-177.740,6.492,148.519
C09848=1196.038,195.393,-58.001,-177.743,6.490,148.519
C09849=1196.043,195.144,-57.978,-177.746,6.488,148.520
C09850=1196.048,194.895,-57.954,-177.749,6.486,148.520
C09851=1196.052,194.647,-57.930,-177.751,6.484,148.520
C09852=1196.057,194.398,-57.907,-177.754,6.482,148.521
C09853=1196.061,194.148,-57.883,-177.756,6.480,148.521
C09854=1196.066,193.899,-57.860,-177.759,6.478,148.521
C09855=1196.070,193.651,-57.836,-177.761,6.476,148.522
C09856=1196.075,193.402,-57.813,-177.764,6.475,148.522
C09857=1196.080,193.153,-57.789,-177.767,6.473,148.522
C09858=1196.085,192.905,-57.766,-177.769,6.471,148.523
C09859=1196.089,192.656,-57.744,-177.772,6.469,148.523
C09860=1196.094,192.407,-57.720,-177.775,6.467,148.523
C09861=1196.098,192.158,-57.696,-177.777,6.465,148.524
C09862=1196.103,191.909,-57.673,-177.780,6.464,148.524
C09863=1196.108,191.660,-57.649,-177.783,6.462,148.524
C09864=1196.112,191.411,-57.626,-177.785,6.460,148.525
C09865=1196.117,191.162,-57.603,-177.788,6.458,148.525
C09866=1196.122,190.913,-57.579,-177.791,6.456,148.525
C09867=1196.126,190.665,-57.557,-177.793,6.454,148.526
C09868=1196.130,190.416,-57.533,-177.795,6.453,148.526
C09869=1196.135,190.167,-57.510,-177.798,6.451,148.526
C09870=1196.140,189.917,-57.487,-177.801,6.449,148.527
C09871=1196.145,189.669,-57.464,-177.803,6.447,148.527
C09872=1196.150,189.420,-57.440,-177.806,6.445,148.527
C09873=1196.153,189.172,-57.417,-177.809,6.443,148.528
C09874=1196.158,188.923,-57.393,-177.811,6.442,148.528
C09875=1196.163,188.674,-57.370,-177.814,6.440,148.528
C09876=1196.168,188.424,-57.347,-177.817,6.438,148.529
C09877=1196.172,188.176,-57.325,-177.819,6.436,148.529
C09878=1196.177,187.927,-57.301,-177.822,6.434,148.529
C09879=1196.182,187.678,-57.278,-177.825,6.433,148.530
C09880=1196.187,187.429,-57.255,-177.827,6.431,148.530
C09881=1196.190,187.180,-57.232,-177.830,6.429,148.531
C09882=1196.195,186.931,-57.209,-177.833,6.427,148.531
C09883=1196.200,186.682,-57.185,-177.835,6.425,148.531
C09884=1196.205,186.433,-57.162,-177.838,6.424,148.532
C09885=1196.209,186.185,-57.139,-177.841,6.422,148.532
C09886=1196.214,185.936,-57.116,-177.843,6.420,148.532
C09887=1196.219,185.687,-57.093,-177.846,6.418,148.533
C09888=1196.223,185.438,-57.071,-177.849,6.416,148.533
C09889=1196.228,185.169,-57.045,-177.851,6.415,148.533
C09890=1196.233,184.899,-57.020,-177.854,6.413,148.534
C09891=1196.238,184.630,-56.996,-177.857,6.411,148.534
C09892=1196.243,184.360,-56.971,-177.859,6.409,148.534
C09893=1196.247,184.111,-56.948,-177.862,6.407,148.535
C09894=1196.252,183.861,-56.925,-177.865,6.406,148.535
C09895=1196.257,183.613,-56.902,-177.867,6.404,148.536
C09896=1196.261,183.364,-56.879,-177.870,6.402,148.536
C09897=1196.266,183.115,-56.856,-177.873,6.400,148.536
C09898=1196.271,182.866,-56.833,-177.875,6.398,148.537
C09899=1196.276,182.618,-56.811,-177.878,6.397,148.537
C09900=1196.280,182.369,-56.788,-177.881,6.395,148.537
C09901=1196.284,182.120,-56.765,-177.883,6.393,148.538
C09902=1196.289,181.870,-56.742,-177.886,6.391,148.538
C09903=1196.293,181.622,-56.719,-177.889,6.389,148.538
C09904=1196.298,181.373,-56.697,-177.891,6.388,148.539
C09905=1196.303,181.124,-56.674,-177.894,6.386,148.539
C09906=1196.307,180.875,-56.651,-177.897,6.384,148.539
C09907=1196.313,180.627,-56.628,-177.899,6.382,148.540
C09908=1196.317,180.377,-56.606,-177.902,6.380,148.540
C09909=1196.322,180.128,-56.583,-177.905,6.379,148.541
C09910=1196.326,179.879,-56.561,-177.907,6.378,148.541
C09911=1196.331,179.630,-56.538,-177.909,6.376,148.541
C09912=1196.335,179.382,-56.515,-177.912,6.374,148.542
C09913=1196.340,179.132,-56.492,-177.915,6.372,148.542
C09914=1196.345,178.884,-56.470,-177.917,6.370,148.542
C09915=1196.350,178.634,-56.447,-177.920,6.369,148.543
C09916=1196.354,178.386,-56.424,-177.923,6.367,148.543
C09917=1196.359,178.136,-56.402,-177.925,6.365,148.543
C09918=1196.363,177.888,-56.379,-177.928,6.363,148.544
C09919=1196.368,177.639,-56.357,-177.931,6.361,148.544
C09920=1196.372,177.390,-56.334,-177.933,6.360,148.544
C09921=1196.377,177.141,-56.312,-177.936,6.358,148.545
C09922=1196.382,176.892,-56.289,-177.939,6.356,148.545
C09923=1196.386,176.643,-56.267,-177.941,6.355,148.546
C09924=1196.391,176.394,-56.244,-177.944,6.354,148.546
C09925=1196.396,176.145,-56.222,-177.947,6.352,148.547
C09926=1196.400,175.897,-56.199,-177.949,6.350,148.547
C09927=1196.405,175.647,-56.177,-177.952,6.348,148.547
C09928=1196.409,175.399,-56.154,-177.955,6.346,148.548
C09929=1196.415,175.150,-56.132,-177.957,6.345,148.548
C09930=1196.419,174.900,-56.110,-177.960,6.343,148.548
C09931=1196.423,174.652,-56.087,-177.963,6.341,148.549
C09932=1196.429,174.403,-56.065,-177.965,6.339,148.549
C09933=1196.433,174.153,-56.043,-177.967,6.338,148.549
C09934=1196.438,173.905,-56.020,-177.970,6.336,148.550
C09935=1196.443,173.656,-55.998,-177.973,6.335,148.550
C09936=1196.447,173.406,-55.976,-177.975,6.333,148.551
C09937=1196.451,173.158,-55.953,-177.978,6.331,148.551
C09938=1196.456,172.909,-55.931,-177.981,6.329,148.551
C09939=1196.461,172.660,-55.909,-177.983,6.327,148.552
C09940=1196.465,172.411,-55.886,-177.986,6.326,148.552
C09941=1196.470,172.162,-55.863,-177.989,6.324,148.553
C09942=1196.475,171.913,-55.842,-177.991,6.323,148.553
C09943=1196.479,171.664,-55.820,-177.994,6.321,148.553
C09944=1196.484,171.416,-55.797,-177.997,6.320,148.554
C09945=1196.489,171.166,-55.775,-177.999,6.318,148.554
C09946=1196.494,170.917,-55.753,-178.002,6.316,148.554
C09947=1196.498,170.668,-55.731,-178.005,6.314,148.555
C09948=1196.503,170.420,-55.709,-178.007,6.313,148.555
C09949=1196.508,170.170,-55.686,-178.010,6.311,148.555
C09950=1196.512,169.922,-55.664,-178.012,6.310,148.556
C09951=1196.517,169.672,-55.642,-178.015,6.308,148.556
C09952=1196.521,169.423,-55.620,-178.017,6.306,148.557
C09953=1196.527,169.174,-55.598,-178.020,6.304,148.557
C09954=1196.531,168.925,-55.576,-178.023,6.303,148.558
C09955=1196.535,168.677,-55.553,-178.026,6.301,148.558
C09956=1196.540,168.427,-55.531,-178.029,6.299,148.558
C09957=1196.545,168.179,-55.510,-178.031,6.298,148.559
C09958=1196.550,167.929,-55.487,-178.033,6.297,148.559
C09959=1196.554,167.680,-55.465,-178.036,6.295,148.559
C09960=1196.559,167.431,-55.443,-178.039,6.293,148.560
C09961=1196.564,167.182,-55.422,-178.041,6.291,148.560
C09962=1196.568,166.934,-55.400,-178.044,6.289,148.561
C09963=1196.573,166.684,-55.378,-178.047,6.288,148.561
C09964=1196.578,166.436,-55.356,-178.049,6.287,148.561
C09965=1196.583,166.186,-55.334,-178.052,6.285,148.562
C09966=1196.587,165.937,-55.312,-178.055,6.283,148.562
C09967=1196.592,165.688,-55.290,-178.057,6.282,148.563
C09968=1196.597,165.440,-55.268,-178.060,6.280,148.563
C09969=1196.601,165.190,-55.246,-178.063,6.278,148.563
C09970=1196.606,164.942,-55.224,-178.065,6.277,148.564
C09971=1196.610,164.692,-55.202,-178.068,6.275,148.564
C09972=1196.615,164.444,-55.181,-178.070,6.273,148.564
C09973=1196.620,164.195,-55.159,-178.073,6.272,148.565
C09974=1196.624,163.946,-55.137,-178.076,6.270,148.565
C09975=1196.629,163.697,-55.115,-178.078,6.269,148.566
C09976=1196.633,163.448,-55.093,-178.081,6.267,148.566
C09977=1196.638,163.199,-55.072,-178.083,6.266,148.567
C09978=1196.643,162.949,-55.050,-178.086,6.264,148.567
C09979=1196.647,162.700,-55.028,-178.089,6.262,148.567
C09980=1196.652,162.452,-55.007,-178.091,6.260,148.568
C09981=1196.657,162.202,-54.985,-178.094,6.260,148.568
C09982=1196.661,161.954,-54.963,-178.097,6.258,148.569
C09983=1196.666,161.704,-54.941,-178.099,6.256,148.569
C09984=1196.671,161.456,-54.919,-178.102,6.254,148.569
C09985=1196.676,161.206,-54.898,-178.105,6.253,148.570
C09986=1196.680,160.957,-54.876,-178.107,6.252,148.570
C09987=1196.685,160.708,-54.855,-178.110,6.250,148.571
C09988=1196.690,160.460,-54.833,-178.113,6.248,148.571
C09989=1196.694,160.210,-54.812,-178.115,6.247,148.571
C09990=1196.699,159.961,-54.790,-178.118,6.245,148.572
C09991=1196.704,159.713,-54.768,-178.120,6.244,148.572
C09992=1196.708,159.463,-54.746,-178.123,6.242,148.573
C09993=1196.714,159.194,-54.723,-178.126,6.240,148.573
C09994=1196.719,158.925,-54.700,-178.129,6.239,148.574
C09995=1196.724,158.656,-54.676,-178.131,6.237,148.574
C09996=1196.729,158.387,-54.653,-178.134,6.235,148.574
//INST
///DATE 2021/06/25 14:28
///ATTR SC,RW,RJ
////FRAME ROBOT
///GROUP1 RB1
NOP
MOVL C00000 V=800.0 PL=0
MOVL C00001 V=800.0 PL=0
MOVL C00002 V=800.0 PL=0
MOVL C00003 V=800.0 PL=0
MOVL C00004 V=800.0 PL=0
MOVL C00005 V=800.0 PL=0
MOVL C00006 V=800.0 PL=0
MOVL C00007 V=800.0 PL=0
MOVL C00008 V=800.0 PL=0
MOVL C00009 V=800.0 PL=0
MOVL C00010 V=800.0 PL=0
MOVL C00011 V=800.0 PL=0
MOVL C00012 V=800.0 PL=0
MOVL C00013 V=800.0 PL=0
MOVL C00014 V=800.0 PL=0
MOVL C00015 V=800.0 PL=0
MOVL C00016 V=800.0 PL=0
MOVL C00017 V=800.0 PL=0
MOVL C00018 V=800.0 PL=0
MOVL C00019 V=800.0 PL=0
MOVL C00020 V=800.0 PL=0
MOVL C00021 V=800.0 PL=0
MOVL C00022 V=800.0 PL=0
MOVL C00023 V=800.0 PL=0
MOVL C00024 V=800.0 PL=0
MOVL C00025 V=800.0 PL=0
MOVL C00026 V=800.0 PL=0
MOVL C00027 V=800.0 PL=0
MOVL C00028 V=800.0 PL=0
MOVL C00029 V=800.0 PL=0
MOVL C00030 V=800.0 PL=0
MOVL C00031 V=800.0 PL=0
MOVL C00032 V=800.0 PL=0
MOVL C00033 V=800.0 PL=0
MOVL C00034 V=800.0 PL=0
MOVL C00035 V=800.0 PL=0
MOVL C00036 V=800.0 PL=0
MOVL C00037 V=800.0 PL=0
MOVL C00038 V=800.0 PL=0
MOVL C00039 V=800.0 PL=0
MOVL C00040 V=800.0 PL=0
MOVL C00041 V=800.0 PL=0
MOVL C00042 V=800.0 PL=0
MOVL C00043 V=800.0 PL=0
MOVL C00044 V=800.0 PL=0
MOVL C00045 V=800.0 PL=0
MOVL C00046 V=800.0 PL=0
MOVL C00047 V=800.0 PL=0
MOVL C00048 V=800.0 PL=0
MOVL C00049 V=800.0 PL=0
MOVL C00050 V=800.0 PL=0
MOVL C00051 V=800.0 PL=0
MOVL C00052 V=800.0 PL=0
MOVL C00053 V=800.0 PL=0
MOVL C00054 V=800.0 PL=0
MOVL C00055 V=800.0 PL=0
MOVL C00056 V=800.0 PL=0
MOVL C00057 V=800.0 PL=0
MOVL C00058 V=800.0 PL=0
MOVL C00059 V=800.0 PL=0
MOVL C00060 V=800.0 PL=0
MOVL C00061 V=800.0 PL=0
MOVL C00062 V=800.0 PL=0
MOVL C00063 V=800.0 PL=0
MOVL C00064 V=800.0 PL=0
MOVL C00065 V=800.0 PL=0
MOVL C00066 V=800.0 PL=0
MOVL C00067 V=800.0 PL=0
MOVL C00068 V=800.0 PL=0
MOVL C00069 V=800.0 PL=0
MOVL C00070 V=800.0 PL=0
MOVL C00071 V=800.0 PL=0
MOVL C00072 V=800.0 PL=0
MOVL C00073 V=800.0 PL=0
MOVL C00074 V=800.0 PL=0
MOVL C00075 V=800.0 PL=0
MOVL C00076 V=800.0 PL=0
MOVL C00077 V=800.0 PL=0
MOVL C00078 V=800.0 PL=0
MOVL C00079 V=800.0 PL=0
MOVL C00080 V=800.0 PL=0
MOVL C00081 V=800.0 PL=0
MOVL C00082 V=800.0 PL=0
MOVL C00083 V=800.0 PL=0
MOVL C00084 V=800.0 PL=0
MOVL C00085 V=800.0 PL=0
MOVL C00086 V=800.0 PL=0
MOVL C00087 V=800.0 PL=0
MOVL C00088 V=800.0 PL=0
MOVL C00089 V=800.0 PL=0
MOVL C00090 V=800.0 PL=0
MOVL C00091 V=800.0 PL=0
MOVL C00092 V=800.0 PL=0
MOVL C00093 V=800.0 PL=0
MOVL C00094 V=800.0 PL=0
MOVL C00095 V=800.0 PL=0
MOVL C00096 V=800.0 PL=0
MOVL C00097 V=800.0 PL=0
MOVL C00098 V=800.0 PL=0
MOVL C00099 V=800.0 PL=0
MOVL C00100 V=800.0 PL=0
MOVL C00101 V=800.0 PL=0
MOVL C00102 V=800.0 PL=0
MOVL C00103 V=800.0 PL=0
MOVL C00104 V=800.0 PL=0
MOVL C00105 V=800.0 PL=0
MOVL C00106 V=800.0 PL=0
MOVL C00107 V=800.0 PL=0
MOVL C00108 V=800.0 PL=0
MOVL C00109 V=800.0 PL=0
MOVL C00110 V=800.0 PL=0
MOVL C00111 V=800.0 PL=0
MOVL C00112 V=800.0 PL=0
MOVL C00113 V=800.0 PL=0
MOVL C00114 V=800.0 PL=0
MOVL C00115 V=800.0 PL=0
MOVL C00116 V=800.0 PL=0
MOVL C00117 V=800.0 PL=0
MOVL C00118 V=800.0 PL=0
MOVL C00119 V=800.0 PL=0
MOVL C00120 V=800.0 PL=0
MOVL C00121 V=800.0 PL=0
MOVL C00122 V=800.0 PL=0
MOVL C00123 V=800.0 PL=0
MOVL C00124 V=800.0 PL=0
MOVL C00125 V=800.0 PL=0
MOVL C00126 V=800.0 PL=0
MOVL C00127 V=800.0 PL=0
MOVL C00128 V=800.0 PL=0
MOVL C00129 V=800.0 PL=0
MOVL C00130 V=800.0 PL=0
MOVL C00131 V=800.0 PL=0
MOVL C00132 V=800.0 PL=0
MOVL C00133 V=800.0 PL=0
MOVL C00134 V=800.0 PL=0
MOVL C00135 V=800.0 PL=0
MOVL C00136 V=800.0 PL=0
MOVL C00137 V=800.0 PL=0
MOVL C00138 V=800.0 PL=0
MOVL C00139 V=800.0 PL=0
MOVL C00140 V=800.0 PL=0
MOVL C00141 V=800.0 PL=0
MOVL C00142 V=800.0 PL=0
MOVL C00143 V=800.0 PL=0
MOVL C00144 V=800.0 PL=0
MOVL C00145 V=800.0 PL=0
MOVL C00146 V=800.0 PL=0
MOVL C00147 V=800.0 PL=0
MOVL C00148 V=800.0 PL=0
MOVL C00149 V=800.0 PL=0
MOVL C00150 V=800.0 PL=0
MOVL C00151 V=800.0 PL=0
MOVL C00152 V=800.0 PL=0
MOVL C00153 V=800.0 PL=0
MOVL C00154 V=800.0 PL=0
MOVL C00155 V=800.0 PL=0
MOVL C00156 V=800.0 PL=0
MOVL C00157 V=800.0 PL=0
MOVL C00158 V=800.0 PL=0
MOVL C00159 V=800.0 PL=0
MOVL C00160 V=800.0 PL=0
MOVL C00161 V=800.0 PL=0
MOVL C00162 V=800.0 PL=0
MOVL C00163 V=800.0 PL=0
MOVL C00164 V=800.0 PL=0
MOVL C00165 V=800.0 PL=0
MOVL C00166 V=800.0 PL=0
MOVL C00167 V=800.0 PL=0
MOVL C00168 V=800.0 PL=0
MOVL C00169 V=800.0 PL=0
MOVL C00170 V=800.0 PL=0
MOVL C00171 V=800.0 PL=0
MOVL C00172 V=800.0 PL=0
MOVL C00173 V=800.0 PL=0
MOVL C00174 V=800.0 PL=0
MOVL C00175 V=800.0 PL=0
MOVL C00176 V=800.0 PL=0
MOVL C00177 V=800.0 PL=0
MOVL C00178 V=800.0 PL=0
MOVL C00179 V=800.0 PL=0
MOVL C00180 V=800.0 PL=0
MOVL C00181 V=800.0 PL=0
MOVL C00182 V=800.0 PL=0
MOVL C00183 V=800.0 PL=0
MOVL C00184 V=800.0 PL=0
MOVL C00185 V=800.0 PL=0
MOVL C00186 V=800.0 PL=0
MOVL C00187 V=800.0 PL=0
MOVL C00188 V=800.0 PL=0
MOVL C00189 V=800.0 PL=0
MOVL C00190 V=800.0 PL=0
MOVL C00191 V=800.0 PL=0
MOVL C00192 V=800.0 PL=0
MOVL C00193 V=800.0 PL=0
MOVL C00194 V=800.0 PL=0
MOVL C00195 V=800.0 PL=0
MOVL C00196 V=800.0 PL=0
MOVL C00197 V=800.0 PL=0
MOVL C00198 V=800.0 PL=0
MOVL C00199 V=800.0 PL=0
MOVL C00200 V=800.0 PL=0
MOVL C00201 V=800.0 PL=0
MOVL C00202 V=800.0 PL=0
MOVL C00203 V=800.0 PL=0
MOVL C00204 V=800.0 PL=0
MOVL C00205 V=800.0 PL=0
MOVL C00206 V=800.0 PL=0
MOVL C00207 V=800.0 PL=0
MOVL C00208 V=800.0 PL=0
MOVL C00209 V=800.0 PL=0
MOVL C00210 V=800.0 PL=0
MOVL C00211 V=800.0 PL=0
MOVL C00212 V=800.0 PL=0
MOVL C00213 V=800.0 PL=0
MOVL C00214 V=800.0 PL=0
MOVL C00215 V=800.0 PL=0
MOVL C00216 V=800.0 PL=0
MOVL C00217 V=800.0 PL=0
MOVL C00218 V=800.0 PL=0
MOVL C00219 V=800.0 PL=0
MOVL C00220 V=800.0 PL=0
MOVL C00221 V=800.0 PL=0
MOVL C00222 V=800.0 PL=0
MOVL C00223 V=800.0 PL=0
MOVL C00224 V=800.0 PL=0
MOVL C00225 V=800.0 PL=0
MOVL C00226 V=800.0 PL=0
MOVL C00227 V=800.0 PL=0
MOVL C00228 V=800.0 PL=0
MOVL C00229 V=800.0 PL=0
MOVL C00230 V=800.0 PL=0
MOVL C00231 V=800.0 PL=0
MOVL C00232 V=800.0 PL=0
MOVL C00233 V=800.0 PL=0
MOVL C00234 V=800.0 PL=0
MOVL C00235 V=800.0 PL=0
MOVL C00236 V=800.0 PL=0
MOVL C00237 V=800.0 PL=0
MOVL C00238 V=800.0 PL=0
MOVL C00239 V=800.0 PL=0
MOVL C00240 V=800.0 PL=0
MOVL C00241 V=800.0 PL=0
MOVL C00242 V=800.0 PL=0
MOVL C00243 V=800.0 PL=0
MOVL C00244 V=800.0 PL=0
MOVL C00245 V=800.0 PL=0
MOVL C00246 V=800.0 PL=0
MOVL C00247 V=800.0 PL=0
MOVL C00248 V=800.0 PL=0
MOVL C00249 V=800.0 PL=0
MOVL C00250 V=800.0 PL=0
MOVL C00251 V=800.0 PL=0
MOVL C00252 V=800.0 PL=0
MOVL C00253 V=800.0 PL=0
MOVL C00254 V=800.0 PL=0
MOVL C00255 V=800.0 PL=0
MOVL C00256 V=800.0 PL=0
MOVL C00257 V=800.0 PL=0
MOVL C00258 V=800.0 PL=0
MOVL C00259 V=800.0 PL=0
MOVL C00260 V=800.0 PL=0
MOVL C00261 V=800.0 PL=0
MOVL C00262 V=800.0 PL=0
MOVL C00263 V=800.0 PL=0
MOVL C00264 V=800.0 PL=0
MOVL C00265 V=800.0 PL=0
MOVL C00266 V=800.0 PL=0
MOVL C00267 V=800.0 PL=0
MOVL C00268 V=800.0 PL=0
MOVL C00269 V=800.0 PL=0
MOVL C00270 V=800.0 PL=0
MOVL C00271 V=800.0 PL=0
MOVL C00272 V=800.0 PL=0
MOVL C00273 V=800.0 PL=0
MOVL C00274 V=800.0 PL=0
MOVL C00275 V=800.0 PL=0
MOVL C00276 V=800.0 PL=0
MOVL C00277 V=800.0 PL=0
MOVL C00278 V=800.0 PL=0
MOVL C00279 V=800.0 PL=0
MOVL C00280 V=800.0 PL=0
MOVL C00281 V=800.0 PL=0
MOVL C00282 V=800.0 PL=0
MOVL C00283 V=800.0 PL=0
MOVL C00284 V=800.0 PL=0
MOVL C00285 V=800.0 PL=0
MOVL C00286 V=800.0 PL=0
MOVL C00287 V=800.0 PL=0
MOVL C00288 V=800.0 PL=0
MOVL C00289 V=800.0 PL=0
MOVL C00290 V=800.0 PL=0
MOVL C00291 V=800.0 PL=0
MOVL C00292 V=800.0 PL=0
MOVL C00293 V=800.0 PL=0
MOVL C00294 V=800.0 PL=0
MOVL C00295 V=800.0 PL=0
MOVL C00296 V=800.0 PL=0
MOVL C00297 V=800.0 PL=0
MOVL C00298 V=800.0 PL=0
MOVL C00299 V=800.0 PL=0
MOVL C00300 V=800.0 PL=0
MOVL C00301 V=800.0 PL=0
MOVL C00302 V=800.0 PL=0
MOVL C00303 V=800.0 PL=0
MOVL C00304 V=800.0 PL=0
MOVL C00305 V=800.0 PL=0
MOVL C00306 V=800.0 PL=0
MOVL C00307 V=800.0 PL=0
MOVL C00308 V=800.0 PL=0
MOVL C00309 V=800.0 PL=0
MOVL C00310 V=800.0 PL=0
MOVL C00311 V=800.0 PL=0
MOVL C00312 V=800.0 PL=0
MOVL C00313 V=800.0 PL=0
MOVL C00314 V=800.0 PL=0
MOVL C00315 V=800.0 PL=0
MOVL C00316 V=800.0 PL=0
MOVL C00317 V=800.0 PL=0
MOVL C00318 V=800.0 PL=0
MOVL C00319 V=800.0 PL=0
MOVL C00320 V=800.0 PL=0
MOVL C00321 V=800.0 PL=0
MOVL C00322 V=800.0 PL=0
MOVL C00323 V=800.0 PL=0
MOVL C00324 V=800.0 PL=0
MOVL C00325 V=800.0 PL=0
MOVL C00326 V=800.0 PL=0
MOVL C00327 V=800.0 PL=0
MOVL C00328 V=800.0 PL=0
MOVL C00329 V=800.0 PL=0
MOVL C00330 V=800.0 PL=0
MOVL C00331 V=800.0 PL=0
MOVL C00332 V=800.0 PL=0
MOVL C00333 V=800.0 PL=0
MOVL C00334 V=800.0 PL=0
MOVL C00335 V=800.0 PL=0
MOVL C00336 V=800.0 PL=0
MOVL C00337 V=800.0 PL=0
MOVL C00338 V=800.0 PL=0
MOVL C00339 V=800.0 PL=0
MOVL C00340 V=800.0 PL=0
MOVL C00341 V=800.0 PL=0
MOVL C00342 V=800.0 PL=0
MOVL C00343 V=800.0 PL=0
MOVL C00344 V=800.0 PL=0
MOVL C00345 V=800.0 PL=0
MOVL C00346 V=800.0 PL=0
MOVL C00347 V=800.0 PL=0
MOVL C00348 V=800.0 PL=0
MOVL C00349 V=800.0 PL=0
MOVL C00350 V=800.0 PL=0
MOVL C00351 V=800.0 PL=0
MOVL C00352 V=800.0 PL=0
MOVL C00353 V=800.0 PL=0
MOVL C00354 V=800.0 PL=0
MOVL C00355 V=800.0 PL=0
MOVL C00356 V=800.0 PL=0
MOVL C00357 V=800.0 PL=0
MOVL C00358 V=800.0 PL=0
MOVL C00359 V=800.0 PL=0
MOVL C00360 V=800.0 PL=0
MOVL C00361 V=800.0 PL=0
MOVL C00362 V=800.0 PL=0
MOVL C00363 V=800.0 PL=0
MOVL C00364 V=800.0 PL=0
MOVL C00365 V=800.0 PL=0
MOVL C00366 V=800.0 PL=0
MOVL C00367 V=800.0 PL=0
MOVL C00368 V=800.0 PL=0
MOVL C00369 V=800.0 PL=0
MOVL C00370 V=800.0 PL=0
MOVL C00371 V=800.0 PL=0
MOVL C00372 V=800.0 PL=0
MOVL C00373 V=800.0 PL=0
MOVL C00374 V=800.0 PL=0
MOVL C00375 V=800.0 PL=0
MOVL C00376 V=800.0 PL=0
MOVL C00377 V=800.0 PL=0
MOVL C00378 V=800.0 PL=0
MOVL C00379 V=800.0 PL=0
MOVL C00380 V=800.0 PL=0
MOVL C00381 V=800.0 PL=0
MOVL C00382 V=800.0 PL=0
MOVL C00383 V=800.0 PL=0
MOVL C00384 V=800.0 PL=0
MOVL C00385 V=800.0 PL=0
MOVL C00386 V=800.0 PL=0
MOVL C00387 V=800.0 PL=0
MOVL C00388 V=800.0 PL=0
MOVL C00389 V=800.0 PL=0
MOVL C00390 V=800.0 PL=0
MOVL C00391 V=800.0 PL=0
MOVL C00392 V=800.0 PL=0
MOVL C00393 V=800.0 PL=0
MOVL C00394 V=800.0 PL=0
MOVL C00395 V=800.0 PL=0
MOVL C00396 V=800.0 PL=0
MOVL C00397 V=800.0 PL=0
MOVL C00398 V=800.0 PL=0
MOVL C00399 V=800.0 PL=0
MOVL C00400 V=800.0 PL=0
MOVL C00401 V=800.0 PL=0
MOVL C00402 V=800.0 PL=0
MOVL C00403 V=800.0 PL=0
MOVL C00404 V=800.0 PL=0
MOVL C00405 V=800.0 PL=0
MOVL C00406 V=800.0 PL=0
MOVL C00407 V=800.0 PL=0
MOVL C00408 V=800.0 PL=0
MOVL C00409 V=800.0 PL=0
MOVL C00410 V=800.0 PL=0
MOVL C00411 V=800.0 PL=0
MOVL C00412 V=800.0 PL=0
MOVL C00413 V=800.0 PL=0
MOVL C00414 V=800.0 PL=0
MOVL C00415 V=800.0 PL=0
MOVL C00416 V=800.0 PL=0
MOVL C00417 V=800.0 PL=0
MOVL C00418 V=800.0 PL=0
MOVL C00419 V=800.0 PL=0
MOVL C00420 V=800.0 PL=0
MOVL C00421 V=800.0 PL=0
MOVL C00422 V=800.0 PL=0
MOVL C00423 V=800.0 PL=0
MOVL C00424 V=800.0 PL=0
MOVL C00425 V=800.0 PL=0
MOVL C00426 V=800.0 PL=0
MOVL C00427 V=800.0 PL=0
MOVL C00428 V=800.0 PL=0
MOVL C00429 V=800.0 PL=0
MOVL C00430 V=800.0 PL=0
MOVL C00431 V=800.0 PL=0
MOVL C00432 V=800.0 PL=0
MOVL C00433 V=800.0 PL=0
MOVL C00434 V=800.0 PL=0
MOVL C00435 V=800.0 PL=0
MOVL C00436 V=800.0 PL=0
MOVL C00437 V=800.0 PL=0
MOVL C00438 V=800.0 PL=0
MOVL C00439 V=800.0 PL=0
MOVL C00440 V=800.0 PL=0
MOVL C00441 V=800.0 PL=0
MOVL C00442 V=800.0 PL=0
MOVL C00443 V=800.0 PL=0
MOVL C00444 V=800.0 PL=0
MOVL C00445 V=800.0 PL=0
MOVL C00446 V=800.0 PL=0
MOVL C00447 V=800.0 PL=0
MOVL C00448 V=800.0 PL=0
MOVL C00449 V=800.0 PL=0
MOVL C00450 V=800.0 PL=0
MOVL C00451 V=800.0 PL=0
MOVL C00452 V=800.0 PL=0
MOVL C00453 V=800.0 PL=0
MOVL C00454 V=800.0 PL=0
MOVL C00455 V=800.0 PL=0
MOVL C00456 V=800.0 PL=0
MOVL C00457 V=800.0 PL=0
MOVL C00458 V=800.0 PL=0
MOVL C00459 V=800.0 PL=0
MOVL C00460 V=800.0 PL=0
MOVL C00461 V=800.0 PL=0
MOVL C00462 V=800.0 PL=0
MOVL C00463 V=800.0 PL=0
MOVL C00464 V=800.0 PL=0
MOVL C00465 V=800.0 PL=0
MOVL C00466 V=800.0 PL=0
MOVL C00467 V=800.0 PL=0
MOVL C00468 V=800.0 PL=0
MOVL C00469 V=800.0 PL=0
MOVL C00470 V=800.0 PL=0
MOVL C00471 V=800.0 PL=0
MOVL C00472 V=800.0 PL=0
MOVL C00473 V=800.0 PL=0
MOVL C00474 V=800.0 PL=0
MOVL C00475 V=800.0 PL=0
MOVL C00476 V=800.0 PL=0
MOVL C00477 V=800.0 PL=0
MOVL C00478 V=800.0 PL=0
MOVL C00479 V=800.0 PL=0
MOVL C00480 V=800.0 PL=0
MOVL C00481 V=800.0 PL=0
MOVL C00482 V=800.0 PL=0
MOVL C00483 V=800.0 PL=0
MOVL C00484 V=800.0 PL=0
MOVL C00485 V=800.0 PL=0
MOVL C00486 V=800.0 PL=0
MOVL C00487 V=800.0 PL=0
MOVL C00488 V=800.0 PL=0
MOVL C00489 V=800.0 PL=0
MOVL C00490 V=800.0 PL=0
MOVL C00491 V=800.0 PL=0
MOVL C00492 V=800.0 PL=0
MOVL C00493 V=800.0 PL=0
MOVL C00494 V=800.0 PL=0
MOVL C00495 V=800.0 PL=0
MOVL C00496 V=800.0 PL=0
MOVL C00497 V=800.0 PL=0
MOVL C00498 V=800.0 PL=0
MOVL C00499 V=800.0 PL=0
MOVL C00500 V=800.0 PL=0
MOVL C00501 V=800.0 PL=0
MOVL C00502 V=800.0 PL=0
MOVL C00503 V=800.0 PL=0
MOVL C00504 V=800.0 PL=0
MOVL C00505 V=800.0 PL=0
MOVL C00506 V=800.0 PL=0
MOVL C00507 V=800.0 PL=0
MOVL C00508 V=800.0 PL=0
MOVL C00509 V=800.0 PL=0
MOVL C00510 V=800.0 PL=0
MOVL C00511 V=800.0 PL=0
MOVL C00512 V=800.0 PL=0
MOVL C00513 V=800.0 PL=0
MOVL C00514 V=800.0 PL=0
MOVL C00515 V=800.0 PL=0
MOVL C00516 V=800.0 PL=0
MOVL C00517 V=800.0 PL=0
MOVL C00518 V=800.0 PL=0
MOVL C00519 V=800.0 PL=0
MOVL C00520 V=800.0 PL=0
MOVL C00521 V=800.0 PL=0
MOVL C00522 V=800.0 PL=0
MOVL C00523 V=800.0 PL=0
MOVL C00524 V=800.0 PL=0
MOVL C00525 V=800.0 PL=0
MOVL C00526 V=800.0 PL=0
MOVL C00527 V=800.0 PL=0
MOVL C00528 V=800.0 PL=0
MOVL C00529 V=800.0 PL=0
MOVL C00530 V=800.0 PL=0
MOVL C00531 V=800.0 PL=0
MOVL C00532 V=800.0 PL=0
MOVL C00533 V=800.0 PL=0
MOVL C00534 V=800.0 PL=0
MOVL C00535 V=800.0 PL=0
MOVL C00536 V=800.0 PL=0
MOVL C00537 V=800.0 PL=0
MOVL C00538 V=800.0 PL=0
MOVL C00539 V=800.0 PL=0
MOVL C00540 V=800.0 PL=0
MOVL C00541 V=800.0 PL=0
MOVL C00542 V=800.0 PL=0
MOVL C00543 V=800.0 PL=0
MOVL C00544 V=800.0 PL=0
MOVL C00545 V=800.0 PL=0
MOVL C00546 V=800.0 PL=0
MOVL C00547 V=800.0 PL=0
MOVL C00548 V=800.0 PL=0
MOVL C00549 V=800.0 PL=0
MOVL C00550 V=800.0 PL=0
MOVL C00551 V=800.0 PL=0
MOVL C00552 V=800.0 PL=0
MOVL C00553 V=800.0 PL=0
MOVL C00554 V=800.0 PL=0
MOVL C00555 V=800.0 PL=0
MOVL C00556 V=800.0 PL=0
MOVL C00557 V=800.0 PL=0
MOVL C00558 V=800.0 PL=0
MOVL C00559 V=800.0 PL=0
MOVL C00560 V=800.0 PL=0
MOVL C00561 V=800.0 PL=0
MOVL C00562 V=800.0 PL=0
MOVL C00563 V=800.0 PL=0
MOVL C00564 V=800.0 PL=0
MOVL C00565 V=800.0 PL=0
MOVL C00566 V=800.0 PL=0
MOVL C00567 V=800.0 PL=0
MOVL C00568 V=800.0 PL=0
MOVL C00569 V=800.0 PL=0
MOVL C00570 V=800.0 PL=0
MOVL C00571 V=800.0 PL=0
MOVL C00572 V=800.0 PL=0
MOVL C00573 V=800.0 PL=0
MOVL C00574 V=800.0 PL=0
MOVL C00575 V=800.0 PL=0
MOVL C00576 V=800.0 PL=0
MOVL C00577 V=800.0 PL=0
MOVL C00578 V=800.0 PL=0
MOVL C00579 V=800.0 PL=0
MOVL C00580 V=800.0 PL=0
MOVL C00581 V=800.0 PL=0
MOVL C00582 V=800.0 PL=0
MOVL C00583 V=800.0 PL=0
MOVL C00584 V=800.0 PL=0
MOVL C00585 V=800.0 PL=0
MOVL C00586 V=800.0 PL=0
MOVL C00587 V=800.0 PL=0
MOVL C00588 V=800.0 PL=0
MOVL C00589 V=800.0 PL=0
MOVL C00590 V=800.0 PL=0
MOVL C00591 V=800.0 PL=0
MOVL C00592 V=800.0 PL=0
MOVL C00593 V=800.0 PL=0
MOVL C00594 V=800.0 PL=0
MOVL C00595 V=800.0 PL=0
MOVL C00596 V=800.0 PL=0
MOVL C00597 V=800.0 PL=0
MOVL C00598 V=800.0 PL=0
MOVL C00599 V=800.0 PL=0
MOVL C00600 V=800.0 PL=0
MOVL C00601 V=800.0 PL=0
MOVL C00602 V=800.0 PL=0
MOVL C00603 V=800.0 PL=0
MOVL C00604 V=800.0 PL=0
MOVL C00605 V=800.0 PL=0
MOVL C00606 V=800.0 PL=0
MOVL C00607 V=800.0 PL=0
MOVL C00608 V=800.0 PL=0
MOVL C00609 V=800.0 PL=0
MOVL C00610 V=800.0 PL=0
MOVL C00611 V=800.0 PL=0
MOVL C00612 V=800.0 PL=0
MOVL C00613 V=800.0 PL=0
MOVL C00614 V=800.0 PL=0
MOVL C00615 V=800.0 PL=0
MOVL C00616 V=800.0 PL=0
MOVL C00617 V=800.0 PL=0
MOVL C00618 V=800.0 PL=0
MOVL C00619 V=800.0 PL=0
MOVL C00620 V=800.0 PL=0
MOVL C00621 V=800.0 PL=0
MOVL C00622 V=800.0 PL=0
MOVL C00623 V=800.0 PL=0
MOVL C00624 V=800.0 PL=0
MOVL C00625 V=800.0 PL=0
MOVL C00626 V=800.0 PL=0
MOVL C00627 V=800.0 PL=0
MOVL C00628 V=800.0 PL=0
MOVL C00629 V=800.0 PL=0
MOVL C00630 V=800.0 PL=0
MOVL C00631 V=800.0 PL=0
MOVL C00632 V=800.0 PL=0
MOVL C00633 V=800.0 PL=0
MOVL C00634 V=800.0 PL=0
MOVL C00635 V=800.0 PL=0
MOVL C00636 V=800.0 PL=0
MOVL C00637 V=800.0 PL=0
MOVL C00638 V=800.0 PL=0
MOVL C00639 V=800.0 PL=0
MOVL C00640 V=800.0 PL=0
MOVL C00641 V=800.0 PL=0
MOVL C00642 V=800.0 PL=0
MOVL C00643 V=800.0 PL=0
MOVL C00644 V=800.0 PL=0
MOVL C00645 V=800.0 PL=0
MOVL C00646 V=800.0 PL=0
MOVL C00647 V=800.0 PL=0
MOVL C00648 V=800.0 PL=0
MOVL C00649 V=800.0 PL=0
MOVL C00650 V=800.0 PL=0
MOVL C00651 V=800.0 PL=0
MOVL C00652 V=800.0 PL=0
MOVL C00653 V=800.0 PL=0
MOVL C00654 V=800.0 PL=0
MOVL C00655 V=800.0 PL=0
MOVL C00656 V=800.0 PL=0
MOVL C00657 V=800.0 PL=0
MOVL C00658 V=800.0 PL=0
MOVL C00659 V=800.0 PL=0
MOVL C00660 V=800.0 PL=0
MOVL C00661 V=800.0 PL=0
MOVL C00662 V=800.0 PL=0
MOVL C00663 V=800.0 PL=0
MOVL C00664 V=800.0 PL=0
MOVL C00665 V=800.0 PL=0
MOVL C00666 V=800.0 PL=0
MOVL C00667 V=800.0 PL=0
MOVL C00668 V=800.0 PL=0
MOVL C00669 V=800.0 PL=0
MOVL C00670 V=800.0 PL=0
MOVL C00671 V=800.0 PL=0
MOVL C00672 V=800.0 PL=0
MOVL C00673 V=800.0 PL=0
MOVL C00674 V=800.0 PL=0
MOVL C00675 V=800.0 PL=0
MOVL C00676 V=800.0 PL=0
MOVL C00677 V=800.0 PL=0
MOVL C00678 V=800.0 PL=0
MOVL C00679 V=800.0 PL=0
MOVL C00680 V=800.0 PL=0
MOVL C00681 V=800.0 PL=0
MOVL C00682 V=800.0 PL=0
MOVL C00683 V=800.0 PL=0
MOVL C00684 V=800.0 PL=0
MOVL C00685 V=800.0 PL=0
MOVL C00686 V=800.0 PL=0
MOVL C00687 V=800.0 PL=0
MOVL C00688 V=800.0 PL=0
MOVL C00689 V=800.0 PL=0
MOVL C00690 V=800.0 PL=0
MOVL C00691 V=800.0 PL=0
MOVL C00692 V=800.0 PL=0
MOVL C00693 V=800.0 PL=0
MOVL C00694 V=800.0 PL=0
MOVL C00695 V=800.0 PL=0
MOVL C00696 V=800.0 PL=0
MOVL C00697 V=800.0 PL=0
MOVL C00698 V=800.0 PL=0
MOVL C00699 V=800.0 PL=0
MOVL C00700 V=800.0 PL=0
MOVL C00701 V=800.0 PL=0
MOVL C00702 V=800.0 PL=0
MOVL C00703 V=800.0 PL=0
MOVL C00704 V=800.0 PL=0
MOVL C00705 V=800.0 PL=0
MOVL C00706 V=800.0 PL=0
MOVL C00707 V=800.0 PL=0
MOVL C00708 V=800.0 PL=0
MOVL C00709 V=800.0 PL=0
MOVL C00710 V=800.0 PL=0
MOVL C00711 V=800.0 PL=0
MOVL C00712 V=800.0 PL=0
MOVL C00713 V=800.0 PL=0
MOVL C00714 V=800.0 PL=0
MOVL C00715 V=800.0 PL=0
MOVL C00716 V=800.0 PL=0
MOVL C00717 V=800.0 PL=0
MOVL C00718 V=800.0 PL=0
MOVL C00719 V=800.0 PL=0
MOVL C00720 V=800.0 PL=0
MOVL C00721 V=800.0 PL=0
MOVL C00722 V=800.0 PL=0
MOVL C00723 V=800.0 PL=0
MOVL C00724 V=800.0 PL=0
MOVL C00725 V=800.0 PL=0
MOVL C00726 V=800.0 PL=0
MOVL C00727 V=800.0 PL=0
MOVL C00728 V=800.0 PL=0
MOVL C00729 V=800.0 PL=0
MOVL C00730 V=800.0 PL=0
MOVL C00731 V=800.0 PL=0
MOVL C00732 V=800.0 PL=0
MOVL C00733 V=800.0 PL=0
MOVL C00734 V=800.0 PL=0
MOVL C00735 V=800.0 PL=0
MOVL C00736 V=800.0 PL=0
MOVL C00737 V=800.0 PL=0
MOVL C00738 V=800.0 PL=0
MOVL C00739 V=800.0 PL=0
MOVL C00740 V=800.0 PL=0
MOVL C00741 V=800.0 PL=0
MOVL C00742 V=800.0 PL=0
MOVL C00743 V=800.0 PL=0
MOVL C00744 V=800.0 PL=0
MOVL C00745 V=800.0 PL=0
MOVL C00746 V=800.0 PL=0
MOVL C00747 V=800.0 PL=0
MOVL C00748 V=800.0 PL=0
MOVL C00749 V=800.0 PL=0
MOVL C00750 V=800.0 PL=0
MOVL C00751 V=800.0 PL=0
MOVL C00752 V=800.0 PL=0
MOVL C00753 V=800.0 PL=0
MOVL C00754 V=800.0 PL=0
MOVL C00755 V=800.0 PL=0
MOVL C00756 V=800.0 PL=0
MOVL C00757 V=800.0 PL=0
MOVL C00758 V=800.0 PL=0
MOVL C00759 V=800.0 PL=0
MOVL C00760 V=800.0 PL=0
MOVL C00761 V=800.0 PL=0
MOVL C00762 V=800.0 PL=0
MOVL C00763 V=800.0 PL=0
MOVL C00764 V=800.0 PL=0
MOVL C00765 V=800.0 PL=0
MOVL C00766 V=800.0 PL=0
MOVL C00767 V=800.0 PL=0
MOVL C00768 V=800.0 PL=0
MOVL C00769 V=800.0 PL=0
MOVL C00770 V=800.0 PL=0
MOVL C00771 V=800.0 PL=0
MOVL C00772 V=800.0 PL=0
MOVL C00773 V=800.0 PL=0
MOVL C00774 V=800.0 PL=0
MOVL C00775 V=800.0 PL=0
MOVL C00776 V=800.0 PL=0
MOVL C00777 V=800.0 PL=0
MOVL C00778 V=800.0 PL=0
MOVL C00779 V=800.0 PL=0
MOVL C00780 V=800.0 PL=0
MOVL C00781 V=800.0 PL=0
MOVL C00782 V=800.0 PL=0
MOVL C00783 V=800.0 PL=0
MOVL C00784 V=800.0 PL=0
MOVL C00785 V=800.0 PL=0
MOVL C00786 V=800.0 PL=0
MOVL C00787 V=800.0 PL=0
MOVL C00788 V=800.0 PL=0
MOVL C00789 V=800.0 PL=0
MOVL C00790 V=800.0 PL=0
MOVL C00791 V=800.0 PL=0
MOVL C00792 V=800.0 PL=0
MOVL C00793 V=800.0 PL=0
MOVL C00794 V=800.0 PL=0
MOVL C00795 V=800.0 PL=0
MOVL C00796 V=800.0 PL=0
MOVL C00797 V=800.0 PL=0
MOVL C00798 V=800.0 PL=0
MOVL C00799 V=800.0 PL=0
MOVL C00800 V=800.0 PL=0
MOVL C00801 V=800.0 PL=0
MOVL C00802 V=800.0 PL=0
MOVL C00803 V=800.0 PL=0
MOVL C00804 V=800.0 PL=0
MOVL C00805 V=800.0 PL=0
MOVL C00806 V=800.0 PL=0
MOVL C00807 V=800.0 PL=0
MOVL C00808 V=800.0 PL=0
MOVL C00809 V=800.0 PL=0
MOVL C00810 V=800.0 PL=0
MOVL C00811 V=800.0 PL=0
MOVL C00812 V=800.0 PL=0
MOVL C00813 V=800.0 PL=0
MOVL C00814 V=800.0 PL=0
MOVL C00815 V=800.0 PL=0
MOVL C00816 V=800.0 PL=0
MOVL C00817 V=800.0 PL=0
MOVL C00818 V=800.0 PL=0
MOVL C00819 V=800.0 PL=0
MOVL C00820 V=800.0 PL=0
MOVL C00821 V=800.0 PL=0
MOVL C00822 V=800.0 PL=0
MOVL C00823 V=800.0 PL=0
MOVL C00824 V=800.0 PL=0
MOVL C00825 V=800.0 PL=0
MOVL C00826 V=800.0 PL=0
MOVL C00827 V=800.0 PL=0
MOVL C00828 V=800.0 PL=0
MOVL C00829 V=800.0 PL=0
MOVL C00830 V=800.0 PL=0
MOVL C00831 V=800.0 PL=0
MOVL C00832 V=800.0 PL=0
MOVL C00833 V=800.0 PL=0
MOVL C00834 V=800.0 PL=0
MOVL C00835 V=800.0 PL=0
MOVL C00836 V=800.0 PL=0
MOVL C00837 V=800.0 PL=0
MOVL C00838 V=800.0 PL=0
MOVL C00839 V=800.0 PL=0
MOVL C00840 V=800.0 PL=0
MOVL C00841 V=800.0 PL=0
MOVL C00842 V=800.0 PL=0
MOVL C00843 V=800.0 PL=0
MOVL C00844 V=800.0 PL=0
MOVL C00845 V=800.0 PL=0
MOVL C00846 V=800.0 PL=0
MOVL C00847 V=800.0 PL=0
MOVL C00848 V=800.0 PL=0
MOVL C00849 V=800.0 PL=0
MOVL C00850 V=800.0 PL=0
MOVL C00851 V=800.0 PL=0
MOVL C00852 V=800.0 PL=0
MOVL C00853 V=800.0 PL=0
MOVL C00854 V=800.0 PL=0
MOVL C00855 V=800.0 PL=0
MOVL C00856 V=800.0 PL=0
MOVL C00857 V=800.0 PL=0
MOVL C00858 V=800.0 PL=0
MOVL C00859 V=800.0 PL=0
MOVL C00860 V=800.0 PL=0
MOVL C00861 V=800.0 PL=0
MOVL C00862 V=800.0 PL=0
MOVL C00863 V=800.0 PL=0
MOVL C00864 V=800.0 PL=0
MOVL C00865 V=800.0 PL=0
MOVL C00866 V=800.0 PL=0
MOVL C00867 V=800.0 PL=0
MOVL C00868 V=800.0 PL=0
MOVL C00869 V=800.0 PL=0
MOVL C00870 V=800.0 PL=0
MOVL C00871 V=800.0 PL=0
MOVL C00872 V=800.0 PL=0
MOVL C00873 V=800.0 PL=0
MOVL C00874 V=800.0 PL=0
MOVL C00875 V=800.0 PL=0
MOVL C00876 V=800.0 PL=0
MOVL C00877 V=800.0 PL=0
MOVL C00878 V=800.0 PL=0
MOVL C00879 V=800.0 PL=0
MOVL C00880 V=800.0 PL=0
MOVL C00881 V=800.0 PL=0
MOVL C00882 V=800.0 PL=0
MOVL C00883 V=800.0 PL=0
MOVL C00884 V=800.0 PL=0
MOVL C00885 V=800.0 PL=0
MOVL C00886 V=800.0 PL=0
MOVL C00887 V=800.0 PL=0
MOVL C00888 V=800.0 PL=0
MOVL C00889 V=800.0 PL=0
MOVL C00890 V=800.0 PL=0
MOVL C00891 V=800.0 PL=0
MOVL C00892 V=800.0 PL=0
MOVL C00893 V=800.0 PL=0
MOVL C00894 V=800.0 PL=0
MOVL C00895 V=800.0 PL=0
MOVL C00896 V=800.0 PL=0
MOVL C00897 V=800.0 PL=0
MOVL C00898 V=800.0 PL=0
MOVL C00899 V=800.0 PL=0
MOVL C00900 V=800.0 PL=0
MOVL C00901 V=800.0 PL=0
MOVL C00902 V=800.0 PL=0
MOVL C00903 V=800.0 PL=0
MOVL C00904 V=800.0 PL=0
MOVL C00905 V=800.0 PL=0
MOVL C00906 V=800.0 PL=0
MOVL C00907 V=800.0 PL=0
MOVL C00908 V=800.0 PL=0
MOVL C00909 V=800.0 PL=0
MOVL C00910 V=800.0 PL=0
MOVL C00911 V=800.0 PL=0
MOVL C00912 V=800.0 PL=0
MOVL C00913 V=800.0 PL=0
MOVL C00914 V=800.0 PL=0
MOVL C00915 V=800.0 PL=0
MOVL C00916 V=800.0 PL=0
MOVL C00917 V=800.0 PL=0
MOVL C00918 V=800.0 PL=0
MOVL C00919 V=800.0 PL=0
MOVL C00920 V=800.0 PL=0
MOVL C00921 V=800.0 PL=0
MOVL C00922 V=800.0 PL=0
MOVL C00923 V=800.0 PL=0
MOVL C00924 V=800.0 PL=0
MOVL C00925 V=800.0 PL=0
MOVL C00926 V=800.0 PL=0
MOVL C00927 V=800.0 PL=0
MOVL C00928 V=800.0 PL=0
MOVL C00929 V=800.0 PL=0
MOVL C00930 V=800.0 PL=0
MOVL C00931 V=800.0 PL=0
MOVL C00932 V=800.0 PL=0
MOVL C00933 V=800.0 PL=0
MOVL C00934 V=800.0 PL=0
MOVL C00935 V=800.0 PL=0
MOVL C00936 V=800.0 PL=0
MOVL C00937 V=800.0 PL=0
MOVL C00938 V=800.0 PL=0
MOVL C00939 V=800.0 PL=0
MOVL C00940 V=800.0 PL=0
MOVL C00941 V=800.0 PL=0
MOVL C00942 V=800.0 PL=0
MOVL C00943 V=800.0 PL=0
MOVL C00944 V=800.0 PL=0
MOVL C00945 V=800.0 PL=0
MOVL C00946 V=800.0 PL=0
MOVL C00947 V=800.0 PL=0
MOVL C00948 V=800.0 PL=0
MOVL C00949 V=800.0 PL=0
MOVL C00950 V=800.0 PL=0
MOVL C00951 V=800.0 PL=0
MOVL C00952 V=800.0 PL=0
MOVL C00953 V=800.0 PL=0
MOVL C00954 V=800.0 PL=0
MOVL C00955 V=800.0 PL=0
MOVL C00956 V=800.0 PL=0
MOVL C00957 V=800.0 PL=0
MOVL C00958 V=800.0 PL=0
MOVL C00959 V=800.0 PL=0
MOVL C00960 V=800.0 PL=0
MOVL C00961 V=800.0 PL=0
MOVL C00962 V=800.0 PL=0
MOVL C00963 V=800.0 PL=0
MOVL C00964 V=800.0 PL=0
MOVL C00965 V=800.0 PL=0
MOVL C00966 V=800.0 PL=0
MOVL C00967 V=800.0 PL=0
MOVL C00968 V=800.0 PL=0
MOVL C00969 V=800.0 PL=0
MOVL C00970 V=800.0 PL=0
MOVL C00971 V=800.0 PL=0
MOVL C00972 V=800.0 PL=0
MOVL C00973 V=800.0 PL=0
MOVL C00974 V=800.0 PL=0
MOVL C00975 V=800.0 PL=0
MOVL C00976 V=800.0 PL=0
MOVL C00977 V=800.0 PL=0
MOVL C00978 V=800.0 PL=0
MOVL C00979 V=800.0 PL=0
MOVL C00980 V=800.0 PL=0
MOVL C00981 V=800.0 PL=0
MOVL C00982 V=800.0 PL=0
MOVL C00983 V=800.0 PL=0
MOVL C00984 V=800.0 PL=0
MOVL C00985 V=800.0 PL=0
MOVL C00986 V=800.0 PL=0
MOVL C00987 V=800.0 PL=0
MOVL C00988 V=800.0 PL=0
MOVL C00989 V=800.0 PL=0
MOVL C00990 V=800.0 PL=0
MOVL C00991 V=800.0 PL=0
MOVL C00992 V=800.0 PL=0
MOVL C00993 V=800.0 PL=0
MOVL C00994 V=800.0 PL=0
MOVL C00995 V=800.0 PL=0
MOVL C00996 V=800.0 PL=0
MOVL C00997 V=800.0 PL=0
MOVL C00998 V=800.0 PL=0
MOVL C00999 V=800.0 PL=0
MOVL C01000 V=800.0 PL=0
MOVL C01001 V=800.0 PL=0
MOVL C01002 V=800.0 PL=0
MOVL C01003 V=800.0 PL=0
MOVL C01004 V=800.0 PL=0
MOVL C01005 V=800.0 PL=0
MOVL C01006 V=800.0 PL=0
MOVL C01007 V=800.0 PL=0
MOVL C01008 V=800.0 PL=0
MOVL C01009 V=800.0 PL=0
MOVL C01010 V=800.0 PL=0
MOVL C01011 V=800.0 PL=0
MOVL C01012 V=800.0 PL=0
MOVL C01013 V=800.0 PL=0
MOVL C01014 V=800.0 PL=0
MOVL C01015 V=800.0 PL=0
MOVL C01016 V=800.0 PL=0
MOVL C01017 V=800.0 PL=0
MOVL C01018 V=800.0 PL=0
MOVL C01019 V=800.0 PL=0
MOVL C01020 V=800.0 PL=0
MOVL C01021 V=800.0 PL=0
MOVL C01022 V=800.0 PL=0
MOVL C01023 V=800.0 PL=0
MOVL C01024 V=800.0 PL=0
MOVL C01025 V=800.0 PL=0
MOVL C01026 V=800.0 PL=0
MOVL C01027 V=800.0 PL=0
MOVL C01028 V=800.0 PL=0
MOVL C01029 V=800.0 PL=0
MOVL C01030 V=800.0 PL=0
MOVL C01031 V=800.0 PL=0
MOVL C01032 V=800.0 PL=0
MOVL C01033 V=800.0 PL=0
MOVL C01034 V=800.0 PL=0
MOVL C01035 V=800.0 PL=0
MOVL C01036 V=800.0 PL=0
MOVL C01037 V=800.0 PL=0
MOVL C01038 V=800.0 PL=0
MOVL C01039 V=800.0 PL=0
MOVL C01040 V=800.0 PL=0
MOVL C01041 V=800.0 PL=0
MOVL C01042 V=800.0 PL=0
MOVL C01043 V=800.0 PL=0
MOVL C01044 V=800.0 PL=0
MOVL C01045 V=800.0 PL=0
MOVL C01046 V=800.0 PL=0
MOVL C01047 V=800.0 PL=0
MOVL C01048 V=800.0 PL=0
MOVL C01049 V=800.0 PL=0
MOVL C01050 V=800.0 PL=0
MOVL C01051 V=800.0 PL=0
MOVL C01052 V=800.0 PL=0
MOVL C01053 V=800.0 PL=0
MOVL C01054 V=800.0 PL=0
MOVL C01055 V=800.0 PL=0
MOVL C01056 V=800.0 PL=0
MOVL C01057 V=800.0 PL=0
MOVL C01058 V=800.0 PL=0
MOVL C01059 V=800.0 PL=0
MOVL C01060 V=800.0 PL=0
MOVL C01061 V=800.0 PL=0
MOVL C01062 V=800.0 PL=0
MOVL C01063 V=800.0 PL=0
MOVL C01064 V=800.0 PL=0
MOVL C01065 V=800.0 PL=0
MOVL C01066 V=800.0 PL=0
MOVL C01067 V=800.0 PL=0
MOVL C01068 V=800.0 PL=0
MOVL C01069 V=800.0 PL=0
MOVL C01070 V=800.0 PL=0
MOVL C01071 V=800.0 PL=0
MOVL C01072 V=800.0 PL=0
MOVL C01073 V=800.0 PL=0
MOVL C01074 V=800.0 PL=0
MOVL C01075 V=800.0 PL=0
MOVL C01076 V=800.0 PL=0
MOVL C01077 V=800.0 PL=0
MOVL C01078 V=800.0 PL=0
MOVL C01079 V=800.0 PL=0
MOVL C01080 V=800.0 PL=0
MOVL C01081 V=800.0 PL=0
MOVL C01082 V=800.0 PL=0
MOVL C01083 V=800.0 PL=0
MOVL C01084 V=800.0 PL=0
MOVL C01085 V=800.0 PL=0
MOVL C01086 V=800.0 PL=0
MOVL C01087 V=800.0 PL=0
MOVL C01088 V=800.0 PL=0
MOVL C01089 V=800.0 PL=0
MOVL C01090 V=800.0 PL=0
MOVL C01091 V=800.0 PL=0
MOVL C01092 V=800.0 PL=0
MOVL C01093 V=800.0 PL=0
MOVL C01094 V=800.0 PL=0
MOVL C01095 V=800.0 PL=0
MOVL C01096 V=800.0 PL=0
MOVL C01097 V=800.0 PL=0
MOVL C01098 V=800.0 PL=0
MOVL C01099 V=800.0 PL=0
MOVL C01100 V=800.0 PL=0
MOVL C01101 V=800.0 PL=0
MOVL C01102 V=800.0 PL=0
MOVL C01103 V=800.0 PL=0
MOVL C01104 V=800.0 PL=0
MOVL C01105 V=800.0 PL=0
MOVL C01106 V=800.0 PL=0
MOVL C01107 V=800.0 PL=0
MOVL C01108 V=800.0 PL=0
MOVL C01109 V=800.0 PL=0
MOVL C01110 V=800.0 PL=0
MOVL C01111 V=800.0 PL=0
MOVL C01112 V=800.0 PL=0
MOVL C01113 V=800.0 PL=0
MOVL C01114 V=800.0 PL=0
MOVL C01115 V=800.0 PL=0
MOVL C01116 V=800.0 PL=0
MOVL C01117 V=800.0 PL=0
MOVL C01118 V=800.0 PL=0
MOVL C01119 V=800.0 PL=0
MOVL C01120 V=800.0 PL=0
MOVL C01121 V=800.0 PL=0
MOVL C01122 V=800.0 PL=0
MOVL C01123 V=800.0 PL=0
MOVL C01124 V=800.0 PL=0
MOVL C01125 V=800.0 PL=0
MOVL C01126 V=800.0 PL=0
MOVL C01127 V=800.0 PL=0
MOVL C01128 V=800.0 PL=0
MOVL C01129 V=800.0 PL=0
MOVL C01130 V=800.0 PL=0
MOVL C01131 V=800.0 PL=0
MOVL C01132 V=800.0 PL=0
MOVL C01133 V=800.0 PL=0
MOVL C01134 V=800.0 PL=0
MOVL C01135 V=800.0 PL=0
MOVL C01136 V=800.0 PL=0
MOVL C01137 V=800.0 PL=0
MOVL C01138 V=800.0 PL=0
MOVL C01139 V=800.0 PL=0
MOVL C01140 V=800.0 PL=0
MOVL C01141 V=800.0 PL=0
MOVL C01142 V=800.0 PL=0
MOVL C01143 V=800.0 PL=0
MOVL C01144 V=800.0 PL=0
MOVL C01145 V=800.0 PL=0
MOVL C01146 V=800.0 PL=0
MOVL C01147 V=800.0 PL=0
MOVL C01148 V=800.0 PL=0
MOVL C01149 V=800.0 PL=0
MOVL C01150 V=800.0 PL=0
MOVL C01151 V=800.0 PL=0
MOVL C01152 V=800.0 PL=0
MOVL C01153 V=800.0 PL=0
MOVL C01154 V=800.0 PL=0
MOVL C01155 V=800.0 PL=0
MOVL C01156 V=800.0 PL=0
MOVL C01157 V=800.0 PL=0
MOVL C01158 V=800.0 PL=0
MOVL C01159 V=800.0 PL=0
MOVL C01160 V=800.0 PL=0
MOVL C01161 V=800.0 PL=0
MOVL C01162 V=800.0 PL=0
MOVL C01163 V=800.0 PL=0
MOVL C01164 V=800.0 PL=0
MOVL C01165 V=800.0 PL=0
MOVL C01166 V=800.0 PL=0
MOVL C01167 V=800.0 PL=0
MOVL C01168 V=800.0 PL=0
MOVL C01169 V=800.0 PL=0
MOVL C01170 V=800.0 PL=0
MOVL C01171 V=800.0 PL=0
MOVL C01172 V=800.0 PL=0
MOVL C01173 V=800.0 PL=0
MOVL C01174 V=800.0 PL=0
MOVL C01175 V=800.0 PL=0
MOVL C01176 V=800.0 PL=0
MOVL C01177 V=800.0 PL=0
MOVL C01178 V=800.0 PL=0
MOVL C01179 V=800.0 PL=0
MOVL C01180 V=800.0 PL=0
MOVL C01181 V=800.0 PL=0
MOVL C01182 V=800.0 PL=0
MOVL C01183 V=800.0 PL=0
MOVL C01184 V=800.0 PL=0
MOVL C01185 V=800.0 PL=0
MOVL C01186 V=800.0 PL=0
MOVL C01187 V=800.0 PL=0
MOVL C01188 V=800.0 PL=0
MOVL C01189 V=800.0 PL=0
MOVL C01190 V=800.0 PL=0
MOVL C01191 V=800.0 PL=0
MOVL C01192 V=800.0 PL=0
MOVL C01193 V=800.0 PL=0
MOVL C01194 V=800.0 PL=0
MOVL C01195 V=800.0 PL=0
MOVL C01196 V=800.0 PL=0
MOVL C01197 V=800.0 PL=0
MOVL C01198 V=800.0 PL=0
MOVL C01199 V=800.0 PL=0
MOVL C01200 V=800.0 PL=0
MOVL C01201 V=800.0 PL=0
MOVL C01202 V=800.0 PL=0
MOVL C01203 V=800.0 PL=0
MOVL C01204 V=800.0 PL=0
MOVL C01205 V=800.0 PL=0
MOVL C01206 V=800.0 PL=0
MOVL C01207 V=800.0 PL=0
MOVL C01208 V=800.0 PL=0
MOVL C01209 V=800.0 PL=0
MOVL C01210 V=800.0 PL=0
MOVL C01211 V=800.0 PL=0
MOVL C01212 V=800.0 PL=0
MOVL C01213 V=800.0 PL=0
MOVL C01214 V=800.0 PL=0
MOVL C01215 V=800.0 PL=0
MOVL C01216 V=800.0 PL=0
MOVL C01217 V=800.0 PL=0
MOVL C01218 V=800.0 PL=0
MOVL C01219 V=800.0 PL=0
MOVL C01220 V=800.0 PL=0
MOVL C01221 V=800.0 PL=0
MOVL C01222 V=800.0 PL=0
MOVL C01223 V=800.0 PL=0
MOVL C01224 V=800.0 PL=0
MOVL C01225 V=800.0 PL=0
MOVL C01226 V=800.0 PL=0
MOVL C01227 V=800.0 PL=0
MOVL C01228 V=800.0 PL=0
MOVL C01229 V=800.0 PL=0
MOVL C01230 V=800.0 PL=0
MOVL C01231 V=800.0 PL=0
MOVL C01232 V=800.0 PL=0
MOVL C01233 V=800.0 PL=0
MOVL C01234 V=800.0 PL=0
MOVL C01235 V=800.0 PL=0
MOVL C01236 V=800.0 PL=0
MOVL C01237 V=800.0 PL=0
MOVL C01238 V=800.0 PL=0
MOVL C01239 V=800.0 PL=0
MOVL C01240 V=800.0 PL=0
MOVL C01241 V=800.0 PL=0
MOVL C01242 V=800.0 PL=0
MOVL C01243 V=800.0 PL=0
MOVL C01244 V=800.0 PL=0
MOVL C01245 V=800.0 PL=0
MOVL C01246 V=800.0 PL=0
MOVL C01247 V=800.0 PL=0
MOVL C01248 V=800.0 PL=0
MOVL C01249 V=800.0 PL=0
MOVL C01250 V=800.0 PL=0
MOVL C01251 V=800.0 PL=0
MOVL C01252 V=800.0 PL=0
MOVL C01253 V=800.0 PL=0
MOVL C01254 V=800.0 PL=0
MOVL C01255 V=800.0 PL=0
MOVL C01256 V=800.0 PL=0
MOVL C01257 V=800.0 PL=0
MOVL C01258 V=800.0 PL=0
MOVL C01259 V=800.0 PL=0
MOVL C01260 V=800.0 PL=0
MOVL C01261 V=800.0 PL=0
MOVL C01262 V=800.0 PL=0
MOVL C01263 V=800.0 PL=0
MOVL C01264 V=800.0 PL=0
MOVL C01265 V=800.0 PL=0
MOVL C01266 V=800.0 PL=0
MOVL C01267 V=800.0 PL=0
MOVL C01268 V=800.0 PL=0
MOVL C01269 V=800.0 PL=0
MOVL C01270 V=800.0 PL=0
MOVL C01271 V=800.0 PL=0
MOVL C01272 V=800.0 PL=0
MOVL C01273 V=800.0 PL=0
MOVL C01274 V=800.0 PL=0
MOVL C01275 V=800.0 PL=0
MOVL C01276 V=800.0 PL=0
MOVL C01277 V=800.0 PL=0
MOVL C01278 V=800.0 PL=0
MOVL C01279 V=800.0 PL=0
MOVL C01280 V=800.0 PL=0
MOVL C01281 V=800.0 PL=0
MOVL C01282 V=800.0 PL=0
MOVL C01283 V=800.0 PL=0
MOVL C01284 V=800.0 PL=0
MOVL C01285 V=800.0 PL=0
MOVL C01286 V=800.0 PL=0
MOVL C01287 V=800.0 PL=0
MOVL C01288 V=800.0 PL=0
MOVL C01289 V=800.0 PL=0
MOVL C01290 V=800.0 PL=0
MOVL C01291 V=800.0 PL=0
MOVL C01292 V=800.0 PL=0
MOVL C01293 V=800.0 PL=0
MOVL C01294 V=800.0 PL=0
MOVL C01295 V=800.0 PL=0
MOVL C01296 V=800.0 PL=0
MOVL C01297 V=800.0 PL=0
MOVL C01298 V=800.0 PL=0
MOVL C01299 V=800.0 PL=0
MOVL C01300 V=800.0 PL=0
MOVL C01301 V=800.0 PL=0
MOVL C01302 V=800.0 PL=0
MOVL C01303 V=800.0 PL=0
MOVL C01304 V=800.0 PL=0
MOVL C01305 V=800.0 PL=0
MOVL C01306 V=800.0 PL=0
MOVL C01307 V=800.0 PL=0
MOVL C01308 V=800.0 PL=0
MOVL C01309 V=800.0 PL=0
MOVL C01310 V=800.0 PL=0
MOVL C01311 V=800.0 PL=0
MOVL C01312 V=800.0 PL=0
MOVL C01313 V=800.0 PL=0
MOVL C01314 V=800.0 PL=0
MOVL C01315 V=800.0 PL=0
MOVL C01316 V=800.0 PL=0
MOVL C01317 V=800.0 PL=0
MOVL C01318 V=800.0 PL=0
MOVL C01319 V=800.0 PL=0
MOVL C01320 V=800.0 PL=0
MOVL C01321 V=800.0 PL=0
MOVL C01322 V=800.0 PL=0
MOVL C01323 V=800.0 PL=0
MOVL C01324 V=800.0 PL=0
MOVL C01325 V=800.0 PL=0
MOVL C01326 V=800.0 PL=0
MOVL C01327 V=800.0 PL=0
MOVL C01328 V=800.0 PL=0
MOVL C01329 V=800.0 PL=0
MOVL C01330 V=800.0 PL=0
MOVL C01331 V=800.0 PL=0
MOVL C01332 V=800.0 PL=0
MOVL C01333 V=800.0 PL=0
MOVL C01334 V=800.0 PL=0
MOVL C01335 V=800.0 PL=0
MOVL C01336 V=800.0 PL=0
MOVL C01337 V=800.0 PL=0
MOVL C01338 V=800.0 PL=0
MOVL C01339 V=800.0 PL=0
MOVL C01340 V=800.0 PL=0
MOVL C01341 V=800.0 PL=0
MOVL C01342 V=800.0 PL=0
MOVL C01343 V=800.0 PL=0
MOVL C01344 V=800.0 PL=0
MOVL C01345 V=800.0 PL=0
MOVL C01346 V=800.0 PL=0
MOVL C01347 V=800.0 PL=0
MOVL C01348 V=800.0 PL=0
MOVL C01349 V=800.0 PL=0
MOVL C01350 V=800.0 PL=0
MOVL C01351 V=800.0 PL=0
MOVL C01352 V=800.0 PL=0
MOVL C01353 V=800.0 PL=0
MOVL C01354 V=800.0 PL=0
MOVL C01355 V=800.0 PL=0
MOVL C01356 V=800.0 PL=0
MOVL C01357 V=800.0 PL=0
MOVL C01358 V=800.0 PL=0
MOVL C01359 V=800.0 PL=0
MOVL C01360 V=800.0 PL=0
MOVL C01361 V=800.0 PL=0
MOVL C01362 V=800.0 PL=0
MOVL C01363 V=800.0 PL=0
MOVL C01364 V=800.0 PL=0
MOVL C01365 V=800.0 PL=0
MOVL C01366 V=800.0 PL=0
MOVL C01367 V=800.0 PL=0
MOVL C01368 V=800.0 PL=0
MOVL C01369 V=800.0 PL=0
MOVL C01370 V=800.0 PL=0
MOVL C01371 V=800.0 PL=0
MOVL C01372 V=800.0 PL=0
MOVL C01373 V=800.0 PL=0
MOVL C01374 V=800.0 PL=0
MOVL C01375 V=800.0 PL=0
MOVL C01376 V=800.0 PL=0
MOVL C01377 V=800.0 PL=0
MOVL C01378 V=800.0 PL=0
MOVL C01379 V=800.0 PL=0
MOVL C01380 V=800.0 PL=0
MOVL C01381 V=800.0 PL=0
MOVL C01382 V=800.0 PL=0
MOVL C01383 V=800.0 PL=0
MOVL C01384 V=800.0 PL=0
MOVL C01385 V=800.0 PL=0
MOVL C01386 V=800.0 PL=0
MOVL C01387 V=800.0 PL=0
MOVL C01388 V=800.0 PL=0
MOVL C01389 V=800.0 PL=0
MOVL C01390 V=800.0 PL=0
MOVL C01391 V=800.0 PL=0
MOVL C01392 V=800.0 PL=0
MOVL C01393 V=800.0 PL=0
MOVL C01394 V=800.0 PL=0
MOVL C01395 V=800.0 PL=0
MOVL C01396 V=800.0 PL=0
MOVL C01397 V=800.0 PL=0
MOVL C01398 V=800.0 PL=0
MOVL C01399 V=800.0 PL=0
MOVL C01400 V=800.0 PL=0
MOVL C01401 V=800.0 PL=0
MOVL C01402 V=800.0 PL=0
MOVL C01403 V=800.0 PL=0
MOVL C01404 V=800.0 PL=0
MOVL C01405 V=800.0 PL=0
MOVL C01406 V=800.0 PL=0
MOVL C01407 V=800.0 PL=0
MOVL C01408 V=800.0 PL=0
MOVL C01409 V=800.0 PL=0
MOVL C01410 V=800.0 PL=0
MOVL C01411 V=800.0 PL=0
MOVL C01412 V=800.0 PL=0
MOVL C01413 V=800.0 PL=0
MOVL C01414 V=800.0 PL=0
MOVL C01415 V=800.0 PL=0
MOVL C01416 V=800.0 PL=0
MOVL C01417 V=800.0 PL=0
MOVL C01418 V=800.0 PL=0
MOVL C01419 V=800.0 PL=0
MOVL C01420 V=800.0 PL=0
MOVL C01421 V=800.0 PL=0
MOVL C01422 V=800.0 PL=0
MOVL C01423 V=800.0 PL=0
MOVL C01424 V=800.0 PL=0
MOVL C01425 V=800.0 PL=0
MOVL C01426 V=800.0 PL=0
MOVL C01427 V=800.0 PL=0
MOVL C01428 V=800.0 PL=0
MOVL C01429 V=800.0 PL=0
MOVL C01430 V=800.0 PL=0
MOVL C01431 V=800.0 PL=0
MOVL C01432 V=800.0 PL=0
MOVL C01433 V=800.0 PL=0
MOVL C01434 V=800.0 PL=0
MOVL C01435 V=800.0 PL=0
MOVL C01436 V=800.0 PL=0
MOVL C01437 V=800.0 PL=0
MOVL C01438 V=800.0 PL=0
MOVL C01439 V=800.0 PL=0
MOVL C01440 V=800.0 PL=0
MOVL C01441 V=800.0 PL=0
MOVL C01442 V=800.0 PL=0
MOVL C01443 V=800.0 PL=0
MOVL C01444 V=800.0 PL=0
MOVL C01445 V=800.0 PL=0
MOVL C01446 V=800.0 PL=0
MOVL C01447 V=800.0 PL=0
MOVL C01448 V=800.0 PL=0
MOVL C01449 V=800.0 PL=0
MOVL C01450 V=800.0 PL=0
MOVL C01451 V=800.0 PL=0
MOVL C01452 V=800.0 PL=0
MOVL C01453 V=800.0 PL=0
MOVL C01454 V=800.0 PL=0
MOVL C01455 V=800.0 PL=0
MOVL C01456 V=800.0 PL=0
MOVL C01457 V=800.0 PL=0
MOVL C01458 V=800.0 PL=0
MOVL C01459 V=800.0 PL=0
MOVL C01460 V=800.0 PL=0
MOVL C01461 V=800.0 PL=0
MOVL C01462 V=800.0 PL=0
MOVL C01463 V=800.0 PL=0
MOVL C01464 V=800.0 PL=0
MOVL C01465 V=800.0 PL=0
MOVL C01466 V=800.0 PL=0
MOVL C01467 V=800.0 PL=0
MOVL C01468 V=800.0 PL=0
MOVL C01469 V=800.0 PL=0
MOVL C01470 V=800.0 PL=0
MOVL C01471 V=800.0 PL=0
MOVL C01472 V=800.0 PL=0
MOVL C01473 V=800.0 PL=0
MOVL C01474 V=800.0 PL=0
MOVL C01475 V=800.0 PL=0
MOVL C01476 V=800.0 PL=0
MOVL C01477 V=800.0 PL=0
MOVL C01478 V=800.0 PL=0
MOVL C01479 V=800.0 PL=0
MOVL C01480 V=800.0 PL=0
MOVL C01481 V=800.0 PL=0
MOVL C01482 V=800.0 PL=0
MOVL C01483 V=800.0 PL=0
MOVL C01484 V=800.0 PL=0
MOVL C01485 V=800.0 PL=0
MOVL C01486 V=800.0 PL=0
MOVL C01487 V=800.0 PL=0
MOVL C01488 V=800.0 PL=0
MOVL C01489 V=800.0 PL=0
MOVL C01490 V=800.0 PL=0
MOVL C01491 V=800.0 PL=0
MOVL C01492 V=800.0 PL=0
MOVL C01493 V=800.0 PL=0
MOVL C01494 V=800.0 PL=0
MOVL C01495 V=800.0 PL=0
MOVL C01496 V=800.0 PL=0
MOVL C01497 V=800.0 PL=0
MOVL C01498 V=800.0 PL=0
MOVL C01499 V=800.0 PL=0
MOVL C01500 V=800.0 PL=0
MOVL C01501 V=800.0 PL=0
MOVL C01502 V=800.0 PL=0
MOVL C01503 V=800.0 PL=0
MOVL C01504 V=800.0 PL=0
MOVL C01505 V=800.0 PL=0
MOVL C01506 V=800.0 PL=0
MOVL C01507 V=800.0 PL=0
MOVL C01508 V=800.0 PL=0
MOVL C01509 V=800.0 PL=0
MOVL C01510 V=800.0 PL=0
MOVL C01511 V=800.0 PL=0
MOVL C01512 V=800.0 PL=0
MOVL C01513 V=800.0 PL=0
MOVL C01514 V=800.0 PL=0
MOVL C01515 V=800.0 PL=0
MOVL C01516 V=800.0 PL=0
MOVL C01517 V=800.0 PL=0
MOVL C01518 V=800.0 PL=0
MOVL C01519 V=800.0 PL=0
MOVL C01520 V=800.0 PL=0
MOVL C01521 V=800.0 PL=0
MOVL C01522 V=800.0 PL=0
MOVL C01523 V=800.0 PL=0
MOVL C01524 V=800.0 PL=0
MOVL C01525 V=800.0 PL=0
MOVL C01526 V=800.0 PL=0
MOVL C01527 V=800.0 PL=0
MOVL C01528 V=800.0 PL=0
MOVL C01529 V=800.0 PL=0
MOVL C01530 V=800.0 PL=0
MOVL C01531 V=800.0 PL=0
MOVL C01532 V=800.0 PL=0
MOVL C01533 V=800.0 PL=0
MOVL C01534 V=800.0 PL=0
MOVL C01535 V=800.0 PL=0
MOVL C01536 V=800.0 PL=0
MOVL C01537 V=800.0 PL=0
MOVL C01538 V=800.0 PL=0
MOVL C01539 V=800.0 PL=0
MOVL C01540 V=800.0 PL=0
MOVL C01541 V=800.0 PL=0
MOVL C01542 V=800.0 PL=0
MOVL C01543 V=800.0 PL=0
MOVL C01544 V=800.0 PL=0
MOVL C01545 V=800.0 PL=0
MOVL C01546 V=800.0 PL=0
MOVL C01547 V=800.0 PL=0
MOVL C01548 V=800.0 PL=0
MOVL C01549 V=800.0 PL=0
MOVL C01550 V=800.0 PL=0
MOVL C01551 V=800.0 PL=0
MOVL C01552 V=800.0 PL=0
MOVL C01553 V=800.0 PL=0
MOVL C01554 V=800.0 PL=0
MOVL C01555 V=800.0 PL=0
MOVL C01556 V=800.0 PL=0
MOVL C01557 V=800.0 PL=0
MOVL C01558 V=800.0 PL=0
MOVL C01559 V=800.0 PL=0
MOVL C01560 V=800.0 PL=0
MOVL C01561 V=800.0 PL=0
MOVL C01562 V=800.0 PL=0
MOVL C01563 V=800.0 PL=0
MOVL C01564 V=800.0 PL=0
MOVL C01565 V=800.0 PL=0
MOVL C01566 V=800.0 PL=0
MOVL C01567 V=800.0 PL=0
MOVL C01568 V=800.0 PL=0
MOVL C01569 V=800.0 PL=0
MOVL C01570 V=800.0 PL=0
MOVL C01571 V=800.0 PL=0
MOVL C01572 V=800.0 PL=0
MOVL C01573 V=800.0 PL=0
MOVL C01574 V=800.0 PL=0
MOVL C01575 V=800.0 PL=0
MOVL C01576 V=800.0 PL=0
MOVL C01577 V=800.0 PL=0
MOVL C01578 V=800.0 PL=0
MOVL C01579 V=800.0 PL=0
MOVL C01580 V=800.0 PL=0
MOVL C01581 V=800.0 PL=0
MOVL C01582 V=800.0 PL=0
MOVL C01583 V=800.0 PL=0
MOVL C01584 V=800.0 PL=0
MOVL C01585 V=800.0 PL=0
MOVL C01586 V=800.0 PL=0
MOVL C01587 V=800.0 PL=0
MOVL C01588 V=800.0 PL=0
MOVL C01589 V=800.0 PL=0
MOVL C01590 V=800.0 PL=0
MOVL C01591 V=800.0 PL=0
MOVL C01592 V=800.0 PL=0
MOVL C01593 V=800.0 PL=0
MOVL C01594 V=800.0 PL=0
MOVL C01595 V=800.0 PL=0
MOVL C01596 V=800.0 PL=0
MOVL C01597 V=800.0 PL=0
MOVL C01598 V=800.0 PL=0
MOVL C01599 V=800.0 PL=0
MOVL C01600 V=800.0 PL=0
MOVL C01601 V=800.0 PL=0
MOVL C01602 V=800.0 PL=0
MOVL C01603 V=800.0 PL=0
MOVL C01604 V=800.0 PL=0
MOVL C01605 V=800.0 PL=0
MOVL C01606 V=800.0 PL=0
MOVL C01607 V=800.0 PL=0
MOVL C01608 V=800.0 PL=0
MOVL C01609 V=800.0 PL=0
MOVL C01610 V=800.0 PL=0
MOVL C01611 V=800.0 PL=0
MOVL C01612 V=800.0 PL=0
MOVL C01613 V=800.0 PL=0
MOVL C01614 V=800.0 PL=0
MOVL C01615 V=800.0 PL=0
MOVL C01616 V=800.0 PL=0
MOVL C01617 V=800.0 PL=0
MOVL C01618 V=800.0 PL=0
MOVL C01619 V=800.0 PL=0
MOVL C01620 V=800.0 PL=0
MOVL C01621 V=800.0 PL=0
MOVL C01622 V=800.0 PL=0
MOVL C01623 V=800.0 PL=0
MOVL C01624 V=800.0 PL=0
MOVL C01625 V=800.0 PL=0
MOVL C01626 V=800.0 PL=0
MOVL C01627 V=800.0 PL=0
MOVL C01628 V=800.0 PL=0
MOVL C01629 V=800.0 PL=0
MOVL C01630 V=800.0 PL=0
MOVL C01631 V=800.0 PL=0
MOVL C01632 V=800.0 PL=0
MOVL C01633 V=800.0 PL=0
MOVL C01634 V=800.0 PL=0
MOVL C01635 V=800.0 PL=0
MOVL C01636 V=800.0 PL=0
MOVL C01637 V=800.0 PL=0
MOVL C01638 V=800.0 PL=0
MOVL C01639 V=800.0 PL=0
MOVL C01640 V=800.0 PL=0
MOVL C01641 V=800.0 PL=0
MOVL C01642 V=800.0 PL=0
MOVL C01643 V=800.0 PL=0
MOVL C01644 V=800.0 PL=0
MOVL C01645 V=800.0 PL=0
MOVL C01646 V=800.0 PL=0
MOVL C01647 V=800.0 PL=0
MOVL C01648 V=800.0 PL=0
MOVL C01649 V=800.0 PL=0
MOVL C01650 V=800.0 PL=0
MOVL C01651 V=800.0 PL=0
MOVL C01652 V=800.0 PL=0
MOVL C01653 V=800.0 PL=0
MOVL C01654 V=800.0 PL=0
MOVL C01655 V=800.0 PL=0
MOVL C01656 V=800.0 PL=0
MOVL C01657 V=800.0 PL=0
MOVL C01658 V=800.0 PL=0
MOVL C01659 V=800.0 PL=0
MOVL C01660 V=800.0 PL=0
MOVL C01661 V=800.0 PL=0
MOVL C01662 V=800.0 PL=0
MOVL C01663 V=800.0 PL=0
MOVL C01664 V=800.0 PL=0
MOVL C01665 V=800.0 PL=0
MOVL C01666 V=800.0 PL=0
MOVL C01667 V=800.0 PL=0
MOVL C01668 V=800.0 PL=0
MOVL C01669 V=800.0 PL=0
MOVL C01670 V=800.0 PL=0
MOVL C01671 V=800.0 PL=0
MOVL C01672 V=800.0 PL=0
MOVL C01673 V=800.0 PL=0
MOVL C01674 V=800.0 PL=0
MOVL C01675 V=800.0 PL=0
MOVL C01676 V=800.0 PL=0
MOVL C01677 V=800.0 PL=0
MOVL C01678 V=800.0 PL=0
MOVL C01679 V=800.0 PL=0
MOVL C01680 V=800.0 PL=0
MOVL C01681 V=800.0 PL=0
MOVL C01682 V=800.0 PL=0
MOVL C01683 V=800.0 PL=0
MOVL C01684 V=800.0 PL=0
MOVL C01685 V=800.0 PL=0
MOVL C01686 V=800.0 PL=0
MOVL C01687 V=800.0 PL=0
MOVL C01688 V=800.0 PL=0
MOVL C01689 V=800.0 PL=0
MOVL C01690 V=800.0 PL=0
MOVL C01691 V=800.0 PL=0
MOVL C01692 V=800.0 PL=0
MOVL C01693 V=800.0 PL=0
MOVL C01694 V=800.0 PL=0
MOVL C01695 V=800.0 PL=0
MOVL C01696 V=800.0 PL=0
MOVL C01697 V=800.0 PL=0
MOVL C01698 V=800.0 PL=0
MOVL C01699 V=800.0 PL=0
MOVL C01700 V=800.0 PL=0
MOVL C01701 V=800.0 PL=0
MOVL C01702 V=800.0 PL=0
MOVL C01703 V=800.0 PL=0
MOVL C01704 V=800.0 PL=0
MOVL C01705 V=800.0 PL=0
MOVL C01706 V=800.0 PL=0
MOVL C01707 V=800.0 PL=0
MOVL C01708 V=800.0 PL=0
MOVL C01709 V=800.0 PL=0
MOVL C01710 V=800.0 PL=0
MOVL C01711 V=800.0 PL=0
MOVL C01712 V=800.0 PL=0
MOVL C01713 V=800.0 PL=0
MOVL C01714 V=800.0 PL=0
MOVL C01715 V=800.0 PL=0
MOVL C01716 V=800.0 PL=0
MOVL C01717 V=800.0 PL=0
MOVL C01718 V=800.0 PL=0
MOVL C01719 V=800.0 PL=0
MOVL C01720 V=800.0 PL=0
MOVL C01721 V=800.0 PL=0
MOVL C01722 V=800.0 PL=0
MOVL C01723 V=800.0 PL=0
MOVL C01724 V=800.0 PL=0
MOVL C01725 V=800.0 PL=0
MOVL C01726 V=800.0 PL=0
MOVL C01727 V=800.0 PL=0
MOVL C01728 V=800.0 PL=0
MOVL C01729 V=800.0 PL=0
MOVL C01730 V=800.0 PL=0
MOVL C01731 V=800.0 PL=0
MOVL C01732 V=800.0 PL=0
MOVL C01733 V=800.0 PL=0
MOVL C01734 V=800.0 PL=0
MOVL C01735 V=800.0 PL=0
MOVL C01736 V=800.0 PL=0
MOVL C01737 V=800.0 PL=0
MOVL C01738 V=800.0 PL=0
MOVL C01739 V=800.0 PL=0
MOVL C01740 V=800.0 PL=0
MOVL C01741 V=800.0 PL=0
MOVL C01742 V=800.0 PL=0
MOVL C01743 V=800.0 PL=0
MOVL C01744 V=800.0 PL=0
MOVL C01745 V=800.0 PL=0
MOVL C01746 V=800.0 PL=0
MOVL C01747 V=800.0 PL=0
MOVL C01748 V=800.0 PL=0
MOVL C01749 V=800.0 PL=0
MOVL C01750 V=800.0 PL=0
MOVL C01751 V=800.0 PL=0
MOVL C01752 V=800.0 PL=0
MOVL C01753 V=800.0 PL=0
MOVL C01754 V=800.0 PL=0
MOVL C01755 V=800.0 PL=0
MOVL C01756 V=800.0 PL=0
MOVL C01757 V=800.0 PL=0
MOVL C01758 V=800.0 PL=0
MOVL C01759 V=800.0 PL=0
MOVL C01760 V=800.0 PL=0
MOVL C01761 V=800.0 PL=0
MOVL C01762 V=800.0 PL=0
MOVL C01763 V=800.0 PL=0
MOVL C01764 V=800.0 PL=0
MOVL C01765 V=800.0 PL=0
MOVL C01766 V=800.0 PL=0
MOVL C01767 V=800.0 PL=0
MOVL C01768 V=800.0 PL=0
MOVL C01769 V=800.0 PL=0
MOVL C01770 V=800.0 PL=0
MOVL C01771 V=800.0 PL=0
MOVL C01772 V=800.0 PL=0
MOVL C01773 V=800.0 PL=0
MOVL C01774 V=800.0 PL=0
MOVL C01775 V=800.0 PL=0
MOVL C01776 V=800.0 PL=0
MOVL C01777 V=800.0 PL=0
MOVL C01778 V=800.0 PL=0
MOVL C01779 V=800.0 PL=0
MOVL C01780 V=800.0 PL=0
MOVL C01781 V=800.0 PL=0
MOVL C01782 V=800.0 PL=0
MOVL C01783 V=800.0 PL=0
MOVL C01784 V=800.0 PL=0
MOVL C01785 V=800.0 PL=0
MOVL C01786 V=800.0 PL=0
MOVL C01787 V=800.0 PL=0
MOVL C01788 V=800.0 PL=0
MOVL C01789 V=800.0 PL=0
MOVL C01790 V=800.0 PL=0
MOVL C01791 V=800.0 PL=0
MOVL C01792 V=800.0 PL=0
MOVL C01793 V=800.0 PL=0
MOVL C01794 V=800.0 PL=0
MOVL C01795 V=800.0 PL=0
MOVL C01796 V=800.0 PL=0
MOVL C01797 V=800.0 PL=0
MOVL C01798 V=800.0 PL=0
MOVL C01799 V=800.0 PL=0
MOVL C01800 V=800.0 PL=0
MOVL C01801 V=800.0 PL=0
MOVL C01802 V=800.0 PL=0
MOVL C01803 V=800.0 PL=0
MOVL C01804 V=800.0 PL=0
MOVL C01805 V=800.0 PL=0
MOVL C01806 V=800.0 PL=0
MOVL C01807 V=800.0 PL=0
MOVL C01808 V=800.0 PL=0
MOVL C01809 V=800.0 PL=0
MOVL C01810 V=800.0 PL=0
MOVL C01811 V=800.0 PL=0
MOVL C01812 V=800.0 PL=0
MOVL C01813 V=800.0 PL=0
MOVL C01814 V=800.0 PL=0
MOVL C01815 V=800.0 PL=0
MOVL C01816 V=800.0 PL=0
MOVL C01817 V=800.0 PL=0
MOVL C01818 V=800.0 PL=0
MOVL C01819 V=800.0 PL=0
MOVL C01820 V=800.0 PL=0
MOVL C01821 V=800.0 PL=0
MOVL C01822 V=800.0 PL=0
MOVL C01823 V=800.0 PL=0
MOVL C01824 V=800.0 PL=0
MOVL C01825 V=800.0 PL=0
MOVL C01826 V=800.0 PL=0
MOVL C01827 V=800.0 PL=0
MOVL C01828 V=800.0 PL=0
MOVL C01829 V=800.0 PL=0
MOVL C01830 V=800.0 PL=0
MOVL C01831 V=800.0 PL=0
MOVL C01832 V=800.0 PL=0
MOVL C01833 V=800.0 PL=0
MOVL C01834 V=800.0 PL=0
MOVL C01835 V=800.0 PL=0
MOVL C01836 V=800.0 PL=0
MOVL C01837 V=800.0 PL=0
MOVL C01838 V=800.0 PL=0
MOVL C01839 V=800.0 PL=0
MOVL C01840 V=800.0 PL=0
MOVL C01841 V=800.0 PL=0
MOVL C01842 V=800.0 PL=0
MOVL C01843 V=800.0 PL=0
MOVL C01844 V=800.0 PL=0
MOVL C01845 V=800.0 PL=0
MOVL C01846 V=800.0 PL=0
MOVL C01847 V=800.0 PL=0
MOVL C01848 V=800.0 PL=0
MOVL C01849 V=800.0 PL=0
MOVL C01850 V=800.0 PL=0
MOVL C01851 V=800.0 PL=0
MOVL C01852 V=800.0 PL=0
MOVL C01853 V=800.0 PL=0
MOVL C01854 V=800.0 PL=0
MOVL C01855 V=800.0 PL=0
MOVL C01856 V=800.0 PL=0
MOVL C01857 V=800.0 PL=0
MOVL C01858 V=800.0 PL=0
MOVL C01859 V=800.0 PL=0
MOVL C01860 V=800.0 PL=0
MOVL C01861 V=800.0 PL=0
MOVL C01862 V=800.0 PL=0
MOVL C01863 V=800.0 PL=0
MOVL C01864 V=800.0 PL=0
MOVL C01865 V=800.0 PL=0
MOVL C01866 V=800.0 PL=0
MOVL C01867 V=800.0 PL=0
MOVL C01868 V=800.0 PL=0
MOVL C01869 V=800.0 PL=0
MOVL C01870 V=800.0 PL=0
MOVL C01871 V=800.0 PL=0
MOVL C01872 V=800.0 PL=0
MOVL C01873 V=800.0 PL=0
MOVL C01874 V=800.0 PL=0
MOVL C01875 V=800.0 PL=0
MOVL C01876 V=800.0 PL=0
MOVL C01877 V=800.0 PL=0
MOVL C01878 V=800.0 PL=0
MOVL C01879 V=800.0 PL=0
MOVL C01880 V=800.0 PL=0
MOVL C01881 V=800.0 PL=0
MOVL C01882 V=800.0 PL=0
MOVL C01883 V=800.0 PL=0
MOVL C01884 V=800.0 PL=0
MOVL C01885 V=800.0 PL=0
MOVL C01886 V=800.0 PL=0
MOVL C01887 V=800.0 PL=0
MOVL C01888 V=800.0 PL=0
MOVL C01889 V=800.0 PL=0
MOVL C01890 V=800.0 PL=0
MOVL C01891 V=800.0 PL=0
MOVL C01892 V=800.0 PL=0
MOVL C01893 V=800.0 PL=0
MOVL C01894 V=800.0 PL=0
MOVL C01895 V=800.0 PL=0
MOVL C01896 V=800.0 PL=0
MOVL C01897 V=800.0 PL=0
MOVL C01898 V=800.0 PL=0
MOVL C01899 V=800.0 PL=0
MOVL C01900 V=800.0 PL=0
MOVL C01901 V=800.0 PL=0
MOVL C01902 V=800.0 PL=0
MOVL C01903 V=800.0 PL=0
MOVL C01904 V=800.0 PL=0
MOVL C01905 V=800.0 PL=0
MOVL C01906 V=800.0 PL=0
MOVL C01907 V=800.0 PL=0
MOVL C01908 V=800.0 PL=0
MOVL C01909 V=800.0 PL=0
MOVL C01910 V=800.0 PL=0
MOVL C01911 V=800.0 PL=0
MOVL C01912 V=800.0 PL=0
MOVL C01913 V=800.0 PL=0
MOVL C01914 V=800.0 PL=0
MOVL C01915 V=800.0 PL=0
MOVL C01916 V=800.0 PL=0
MOVL C01917 V=800.0 PL=0
MOVL C01918 V=800.0 PL=0
MOVL C01919 V=800.0 PL=0
MOVL C01920 V=800.0 PL=0
MOVL C01921 V=800.0 PL=0
MOVL C01922 V=800.0 PL=0
MOVL C01923 V=800.0 PL=0
MOVL C01924 V=800.0 PL=0
MOVL C01925 V=800.0 PL=0
MOVL C01926 V=800.0 PL=0
MOVL C01927 V=800.0 PL=0
MOVL C01928 V=800.0 PL=0
MOVL C01929 V=800.0 PL=0
MOVL C01930 V=800.0 PL=0
MOVL C01931 V=800.0 PL=0
MOVL C01932 V=800.0 PL=0
MOVL C01933 V=800.0 PL=0
MOVL C01934 V=800.0 PL=0
MOVL C01935 V=800.0 PL=0
MOVL C01936 V=800.0 PL=0
MOVL C01937 V=800.0 PL=0
MOVL C01938 V=800.0 PL=0
MOVL C01939 V=800.0 PL=0
MOVL C01940 V=800.0 PL=0
MOVL C01941 V=800.0 PL=0
MOVL C01942 V=800.0 PL=0
MOVL C01943 V=800.0 PL=0
MOVL C01944 V=800.0 PL=0
MOVL C01945 V=800.0 PL=0
MOVL C01946 V=800.0 PL=0
MOVL C01947 V=800.0 PL=0
MOVL C01948 V=800.0 PL=0
MOVL C01949 V=800.0 PL=0
MOVL C01950 V=800.0 PL=0
MOVL C01951 V=800.0 PL=0
MOVL C01952 V=800.0 PL=0
MOVL C01953 V=800.0 PL=0
MOVL C01954 V=800.0 PL=0
MOVL C01955 V=800.0 PL=0
MOVL C01956 V=800.0 PL=0
MOVL C01957 V=800.0 PL=0
MOVL C01958 V=800.0 PL=0
MOVL C01959 V=800.0 PL=0
MOVL C01960 V=800.0 PL=0
MOVL C01961 V=800.0 PL=0
MOVL C01962 V=800.0 PL=0
MOVL C01963 V=800.0 PL=0
MOVL C01964 V=800.0 PL=0
MOVL C01965 V=800.0 PL=0
MOVL C01966 V=800.0 PL=0
MOVL C01967 V=800.0 PL=0
MOVL C01968 V=800.0 PL=0
MOVL C01969 V=800.0 PL=0
MOVL C01970 V=800.0 PL=0
MOVL C01971 V=800.0 PL=0
MOVL C01972 V=800.0 PL=0
MOVL C01973 V=800.0 PL=0
MOVL C01974 V=800.0 PL=0
MOVL C01975 V=800.0 PL=0
MOVL C01976 V=800.0 PL=0
MOVL C01977 V=800.0 PL=0
MOVL C01978 V=800.0 PL=0
MOVL C01979 V=800.0 PL=0
MOVL C01980 V=800.0 PL=0
MOVL C01981 V=800.0 PL=0
MOVL C01982 V=800.0 PL=0
MOVL C01983 V=800.0 PL=0
MOVL C01984 V=800.0 PL=0
MOVL C01985 V=800.0 PL=0
MOVL C01986 V=800.0 PL=0
MOVL C01987 V=800.0 PL=0
MOVL C01988 V=800.0 PL=0
MOVL C01989 V=800.0 PL=0
MOVL C01990 V=800.0 PL=0
MOVL C01991 V=800.0 PL=0
MOVL C01992 V=800.0 PL=0
MOVL C01993 V=800.0 PL=0
MOVL C01994 V=800.0 PL=0
MOVL C01995 V=800.0 PL=0
MOVL C01996 V=800.0 PL=0
MOVL C01997 V=800.0 PL=0
MOVL C01998 V=800.0 PL=0
MOVL C01999 V=800.0 PL=0
MOVL C02000 V=800.0 PL=0
MOVL C02001 V=800.0 PL=0
MOVL C02002 V=800.0 PL=0
MOVL C02003 V=800.0 PL=0
MOVL C02004 V=800.0 PL=0
MOVL C02005 V=800.0 PL=0
MOVL C02006 V=800.0 PL=0
MOVL C02007 V=800.0 PL=0
MOVL C02008 V=800.0 PL=0
MOVL C02009 V=800.0 PL=0
MOVL C02010 V=800.0 PL=0
MOVL C02011 V=800.0 PL=0
MOVL C02012 V=800.0 PL=0
MOVL C02013 V=800.0 PL=0
MOVL C02014 V=800.0 PL=0
MOVL C02015 V=800.0 PL=0
MOVL C02016 V=800.0 PL=0
MOVL C02017 V=800.0 PL=0
MOVL C02018 V=800.0 PL=0
MOVL C02019 V=800.0 PL=0
MOVL C02020 V=800.0 PL=0
MOVL C02021 V=800.0 PL=0
MOVL C02022 V=800.0 PL=0
MOVL C02023 V=800.0 PL=0
MOVL C02024 V=800.0 PL=0
MOVL C02025 V=800.0 PL=0
MOVL C02026 V=800.0 PL=0
MOVL C02027 V=800.0 PL=0
MOVL C02028 V=800.0 PL=0
MOVL C02029 V=800.0 PL=0
MOVL C02030 V=800.0 PL=0
MOVL C02031 V=800.0 PL=0
MOVL C02032 V=800.0 PL=0
MOVL C02033 V=800.0 PL=0
MOVL C02034 V=800.0 PL=0
MOVL C02035 V=800.0 PL=0
MOVL C02036 V=800.0 PL=0
MOVL C02037 V=800.0 PL=0
MOVL C02038 V=800.0 PL=0
MOVL C02039 V=800.0 PL=0
MOVL C02040 V=800.0 PL=0
MOVL C02041 V=800.0 PL=0
MOVL C02042 V=800.0 PL=0
MOVL C02043 V=800.0 PL=0
MOVL C02044 V=800.0 PL=0
MOVL C02045 V=800.0 PL=0
MOVL C02046 V=800.0 PL=0
MOVL C02047 V=800.0 PL=0
MOVL C02048 V=800.0 PL=0
MOVL C02049 V=800.0 PL=0
MOVL C02050 V=800.0 PL=0
MOVL C02051 V=800.0 PL=0
MOVL C02052 V=800.0 PL=0
MOVL C02053 V=800.0 PL=0
MOVL C02054 V=800.0 PL=0
MOVL C02055 V=800.0 PL=0
MOVL C02056 V=800.0 PL=0
MOVL C02057 V=800.0 PL=0
MOVL C02058 V=800.0 PL=0
MOVL C02059 V=800.0 PL=0
MOVL C02060 V=800.0 PL=0
MOVL C02061 V=800.0 PL=0
MOVL C02062 V=800.0 PL=0
MOVL C02063 V=800.0 PL=0
MOVL C02064 V=800.0 PL=0
MOVL C02065 V=800.0 PL=0
MOVL C02066 V=800.0 PL=0
MOVL C02067 V=800.0 PL=0
MOVL C02068 V=800.0 PL=0
MOVL C02069 V=800.0 PL=0
MOVL C02070 V=800.0 PL=0
MOVL C02071 V=800.0 PL=0
MOVL C02072 V=800.0 PL=0
MOVL C02073 V=800.0 PL=0
MOVL C02074 V=800.0 PL=0
MOVL C02075 V=800.0 PL=0
MOVL C02076 V=800.0 PL=0
MOVL C02077 V=800.0 PL=0
MOVL C02078 V=800.0 PL=0
MOVL C02079 V=800.0 PL=0
MOVL C02080 V=800.0 PL=0
MOVL C02081 V=800.0 PL=0
MOVL C02082 V=800.0 PL=0
MOVL C02083 V=800.0 PL=0
MOVL C02084 V=800.0 PL=0
MOVL C02085 V=800.0 PL=0
MOVL C02086 V=800.0 PL=0
MOVL C02087 V=800.0 PL=0
MOVL C02088 V=800.0 PL=0
MOVL C02089 V=800.0 PL=0
MOVL C02090 V=800.0 PL=0
MOVL C02091 V=800.0 PL=0
MOVL C02092 V=800.0 PL=0
MOVL C02093 V=800.0 PL=0
MOVL C02094 V=800.0 PL=0
MOVL C02095 V=800.0 PL=0
MOVL C02096 V=800.0 PL=0
MOVL C02097 V=800.0 PL=0
MOVL C02098 V=800.0 PL=0
MOVL C02099 V=800.0 PL=0
MOVL C02100 V=800.0 PL=0
MOVL C02101 V=800.0 PL=0
MOVL C02102 V=800.0 PL=0
MOVL C02103 V=800.0 PL=0
MOVL C02104 V=800.0 PL=0
MOVL C02105 V=800.0 PL=0
